LIN {X 0,Y 458.169,Z 588.59,A -85,B 0,C 180,E1 7423.789,E2 7423.789} C_VEL
LIN {X 0,Y 488.022,Z 647.13,A -85,B 0,C 180,E1 7427.64,E2 7427.64} C_VEL
LIN {X 0,Y 484.571,Z 716.932,A -85,B 0,C 180,E1 7429.58,E2 7429.58} C_VEL
LIN {X 0,Y 482.25,Z 744.899,A -85,B 0,C 180,E1 7430.929,E2 7430.929} C_VEL
LIN {X 0,Y 471.654,Z 776.533,A -85,B 0,C 180,E1 7432.394,E2 7432.394} C_VEL
LIN {X 0,Y 464.086,Z 836.053,A -85,B 0,C 180,E1 7437.824,E2 7437.824} C_VEL
LIN {X 0,Y 457.551,Z 880.34,A -85,B 0,C 180,E1 7444.194,E2 7444.194} C_VEL
LIN {X 0,Y 453.181,Z 916.717,A -85,B 0,C 180,E1 7452.427,E2 7452.427} C_VEL
LIN {X 0,Y 451.592,Z 937.285,A -85,B 0,C 180,E1 7460.326,E2 7460.326} C_VEL
LIN {X 0,Y 451.133,Z 945.148,A -85,B 0,C 180,E1 7467.107,E2 7467.107} C_VEL
LIN {X 0,Y 451.005,Z 943.768,A -85,B 0,C 180,E1 7474.824,E2 7474.824} C_VEL
LIN {X 0,Y 451.477,Z 931.075,A -85,B 0,C 180,E1 7482.619,E2 7482.619} C_VEL
LIN {X 0,Y 453.83,Z 905.664,A -85,B 0,C 180,E1 7490.554,E2 7490.554} C_VEL
LIN {X 0,Y 459.576,Z 865.156,A -85,B 0,C 180,E1 7498.336,E2 7498.336} C_VEL
LIN {X 0,Y 466.177,Z 818.816,A -85,B 0,C 180,E1 7503.99,E2 7503.99} C_VEL
LIN {X 0,Y 473.707,Z 757.778,A -85,B 0,C 180,E1 7508.771,E2 7508.771} C_VEL
LIN {X 0,Y 479.303,Z 694.506,A -85,B 0,C 180,E1 7511.694,E2 7511.694} C_VEL
LIN {X 0,Y 479.541,Z 644.153,A -85,B 0,C 180,E1 7512.988,E2 7512.988} C_VEL
LIN {X 0,Y 450.022,Z 586.94,A -85,B 0,C 180,E1 7516.817,E2 7516.817} C_VEL
LIN {X 0,Y 449.877,Z 586.94,A -85,B 0,C 180,E1 7526.24,E2 7526.24} C_VEL
LIN {X 0,Y 450.009,Z 586.94,A -85,B 0,C 180,E1 7535.12,E2 7535.12} C_VEL
LIN {X 0,Y 450.376,Z 586.94,A -85,B 0,C 180,E1 7545.406,E2 7545.406} C_VEL
LIN {X 0,Y 450.772,Z 586.94,A -85,B 0,C 180,E1 7555.211,E2 7555.211} C_VEL
LIN {X 0,Y 450.81,Z 586.94,A -85,B 0,C 180,E1 7562.93,E2 7562.93} C_VEL
LIN {X 0,Y 450.783,Z 586.94,A -85,B 0,C 180,E1 7572.672,E2 7572.672} C_VEL
LIN {X 0,Y 450.312,Z 586.94,A -85,B 0,C 180,E1 7582.832,E2 7582.832} C_VEL
LIN {X 0,Y 450.247,Z 588.263,A -85,B 0,C 180,E1 7593.002,E2 7593.002} C_VEL
LIN {X 0,Y 470.605,Z 632.247,A -85,B 0,C 180,E1 7595.934,E2 7595.934} C_VEL
LIN {X 0,Y 466.774,Z 687.738,A -85,B 0,C 180,E1 7598.161,E2 7598.161} C_VEL
LIN {X 0,Y 461.298,Z 735.974,A -85,B 0,C 180,E1 7602.044,E2 7602.044} C_VEL
LIN {X 0,Y 456.216,Z 774.865,A -85,B 0,C 180,E1 7607.473,E2 7607.473} C_VEL
LIN {X 0,Y 452.907,Z 801.492,A -85,B 0,C 180,E1 7614.102,E2 7614.102} C_VEL
LIN {X 0,Y 451.768,Z 813.36,A -85,B 0,C 180,E1 7620.853,E2 7620.853} C_VEL
LIN {X 0,Y 451.997,Z 812.735,A -85,B 0,C 180,E1 7627.45,E2 7627.45} C_VEL
LIN {X 0,Y 453.416,Z 798.561,A -85,B 0,C 180,E1 7634.471,E2 7634.471} C_VEL
LIN {X 0,Y 456.497,Z 770.469,A -85,B 0,C 180,E1 7640.916,E2 7640.916} C_VEL
LIN {X 0,Y 461.148,Z 730.969,A -85,B 0,C 180,E1 7646.109,E2 7646.109} C_VEL
LIN {X 0,Y 466.131,Z 680.829,A -85,B 0,C 180,E1 7649.884,E2 7649.884} C_VEL
LIN {X 0,Y 467.715,Z 623.987,A -85,B 0,C 180,E1 7652.015,E2 7652.015} C_VEL
LIN {X 0,Y 450.876,Z 586.94,A -85,B 0,C 180,E1 7654.344,E2 7654.344} C_VEL
LIN {X 0,Y 450.69,Z 586.94,A -85,B 0,C 180,E1 7664.628,E2 7664.628} C_VEL
LIN {X 0,Y 450.352,Z 586.94,A -85,B 0,C 180,E1 7674.912,E2 7674.912} C_VEL
LIN {X 0,Y 449.926,Z 586.94,A -85,B 0,C 180,E1 7684.243,E2 7684.243} C_VEL
LIN {X 0,Y 449.97,Z 586.94,A -85,B 0,C 180,E1 7693.739,E2 7693.739} C_VEL
LIN {X 0,Y 449.887,Z 586.94,A -85,B 0,C 180,E1 7703.793,E2 7703.793} C_VEL
LIN {X 0,Y 450.197,Z 586.94,A -85,B 0,C 180,E1 7713.288,E2 7713.288} C_VEL
LIN {X 0,Y 450.998,Z 586.94,A -85,B 0,C 180,E1 7725.351,E2 7725.351} C_VEL
LIN {X 0,Y 451.054,Z 586.94,A -85,B 0,C 180,E1 7735.14,E2 7735.14} C_VEL
LIN {X 0,Y 451.103,Z 586.94,A -85,B 0,C 180,E1 7742.854,E2 7742.854} C_VEL
LIN {X 0,Y 450.686,Z 586.94,A -85,B 0,C 180,E1 7752.599,E2 7752.599} C_VEL
LIN {X 0,Y 450.38,Z 586.94,A -85,B 0,C 180,E1 7762.748,E2 7762.748} C_VEL
LIN {X 0,Y 450.056,Z 586.94,A -85,B 0,C 180,E1 7771.452,E2 7771.452} C_VEL
LIN {X 0,Y 449.934,Z 586.94,A -85,B 0,C 180,E1 7781.055,E2 7781.055} C_VEL
LIN {X 0,Y 450.228,Z 588.983,A -85,B 0,C 180,E1 7782.975,E2 7782.975} C_VEL
LIN {X 0,Y 481.575,Z 650.873,A -85,B 0,C 180,E1 7787.149,E2 7787.149} C_VEL
LIN {X 0,Y 477.658,Z 720.311,A -85,B 0,C 180,E1 7789.193,E2 7789.193} C_VEL
LIN {X 0,Y 471.654,Z 776.533,A -85,B 0,C 180,E1 7792.394,E2 7792.394} C_VEL
LIN {X 0,Y 460.687,Z 806.318,A -85,B 0,C 180,E1 7794.355,E2 7794.355} C_VEL
LIN {X 0,Y 452.816,Z 861.229,A -85,B 0,C 180,E1 7800.634,E2 7800.634} C_VEL
LIN {X 0,Y 446.871,Z 900.269,A -85,B 0,C 180,E1 7807.802,E2 7807.802} C_VEL
LIN {X 0,Y 443.887,Z 927.251,A -85,B 0,C 180,E1 7815.616,E2 7815.616} C_VEL
LIN {X 0,Y 442.997,Z 941.682,A -85,B 0,C 180,E1 7823.113,E2 7823.113} C_VEL
LIN {X 0,Y 442.951,Z 945.837,A -85,B 0,C 180,E1 7830.981,E2 7830.981} C_VEL
LIN {X 0,Y 443.529,Z 938.888,A -85,B 0,C 180,E1 7838.856,E2 7838.856} C_VEL
LIN {X 0,Y 444.91,Z 918.74,A -85,B 0,C 180,E1 7847.306,E2 7847.306} C_VEL
LIN {X 0,Y 449.421,Z 883.452,A -85,B 0,C 180,E1 7855.689,E2 7855.689} C_VEL
LIN {X 0,Y 455.739,Z 841.528,A -85,B 0,C 180,E1 7861.897,E2 7861.897} C_VEL
LIN {X 0,Y 463.694,Z 782.474,A -85,B 0,C 180,E1 7867.571,E2 7867.571} C_VEL
LIN {X 0,Y 470.428,Z 717.472,A -85,B 0,C 180,E1 7871.397,E2 7871.397} C_VEL
LIN {X 0,Y 473.618,Z 648.362,A -85,B 0,C 180,E1 7873.423,E2 7873.423} C_VEL
LIN {X 0,Y 441.953,Z 586.94,A -85,B 0,C 180,E1 7877.646,E2 7877.646} C_VEL
LIN {X 0,Y 441.888,Z 586.94,A -85,B 0,C 180,E1 7887.898,E2 7887.898} C_VEL
LIN {X 0,Y 441.894,Z 586.94,A -85,B 0,C 180,E1 7896.789,E2 7896.789} C_VEL
LIN {X 0,Y 442.383,Z 586.94,A -85,B 0,C 180,E1 7907.16,E2 7907.16} C_VEL
LIN {X 0,Y 443.061,Z 586.94,A -85,B 0,C 180,E1 7917.094,E2 7917.094} C_VEL
LIN {X 0,Y 442.991,Z 586.94,A -85,B 0,C 180,E1 7926.921,E2 7926.921} C_VEL
LIN {X 0,Y 442.517,Z 586.94,A -85,B 0,C 180,E1 7936.979,E2 7936.979} C_VEL
LIN {X 0,Y 442.148,Z 586.94,A -85,B 0,C 180,E1 7947.633,E2 7947.633} C_VEL
LIN {X 0,Y 442.299,Z 588.447,A -85,B 0,C 180,E1 7952.157,E2 7952.157} C_VEL
LIN {X 0,Y 464.097,Z 633.334,A -85,B 0,C 180,E1 7955.381,E2 7955.381} C_VEL
LIN {X 0,Y 460.025,Z 688.479,A -85,B 0,C 180,E1 7957.637,E2 7957.637} C_VEL
LIN {X 0,Y 454.191,Z 736.885,A -85,B 0,C 180,E1 7961.585,E2 7961.585} C_VEL
LIN {X 0,Y 448.669,Z 776.328,A -85,B 0,C 180,E1 7967.192,E2 7967.192} C_VEL
LIN {X 0,Y 445.116,Z 802.915,A -85,B 0,C 180,E1 7973.971,E2 7973.971} C_VEL
LIN {X 0,Y 443.913,Z 814.525,A -85,B 0,C 180,E1 7980.695,E2 7980.695} C_VEL
LIN {X 0,Y 444.163,Z 813.367,A -85,B 0,C 180,E1 7988.071,E2 7988.071} C_VEL
LIN {X 0,Y 445.751,Z 798.121,A -85,B 0,C 180,E1 7995.208,E2 7995.208} C_VEL
LIN {X 0,Y 449.244,Z 768.674,A -85,B 0,C 180,E1 8001.747,E2 8001.747} C_VEL
LIN {X 0,Y 454.399,Z 728.304,A -85,B 0,C 180,E1 8006.89,E2 8006.89} C_VEL
LIN {X 0,Y 459.473,Z 677.695,A -85,B 0,C 180,E1 8010.592,E2 8010.592} C_VEL
LIN {X 0,Y 460.9,Z 626.072,A -85,B 0,C 180,E1 8012.536,E2 8012.536} C_VEL
LIN {X 0,Y 442.845,Z 586.94,A -85,B 0,C 180,E1 8015.125,E2 8015.125} C_VEL
LIN {X 0,Y 442.689,Z 586.94,A -85,B 0,C 180,E1 8024.899,E2 8024.899} C_VEL
LIN {X 0,Y 442.304,Z 586.94,A -85,B 0,C 180,E1 8035.397,E2 8035.397} C_VEL
LIN {X 0,Y 441.879,Z 586.94,A -85,B 0,C 180,E1 8046.159,E2 8046.159} C_VEL
LIN {X 0,Y 441.882,Z 586.94,A -85,B 0,C 180,E1 8055.22,E2 8055.22} C_VEL
LIN {X 0,Y 441.938,Z 586.94,A -85,B 0,C 180,E1 8065.458,E2 8065.458} C_VEL
LIN {X 0,Y 442.043,Z 586.94,A -85,B 0,C 180,E1 8075.471,E2 8075.471} C_VEL
LIN {X 0,Y 442.944,Z 586.94,A -85,B 0,C 180,E1 8085.078,E2 8085.078} C_VEL
LIN {X 0,Y 443.054,Z 586.94,A -85,B 0,C 180,E1 8095.052,E2 8095.052} C_VEL
LIN {X 0,Y 443.099,Z 586.94,A -85,B 0,C 180,E1 8102.906,E2 8102.906} C_VEL
LIN {X 0,Y 442.681,Z 586.94,A -85,B 0,C 180,E1 8112.831,E2 8112.831} C_VEL
LIN {X 0,Y 442.32,Z 586.94,A -85,B 0,C 180,E1 8123.187,E2 8123.187} C_VEL
LIN {X 0,Y 441.89,Z 586.94,A -85,B 0,C 180,E1 8132.714,E2 8132.714} C_VEL
LIN {X 0,Y 441.959,Z 587.932,A -85,B 0,C 180,E1 8142.056,E2 8142.056} C_VEL
LIN {X 0,Y 475.063,Z 653.403,A -85,B 0,C 180,E1 8146.623,E2 8146.623} C_VEL
LIN {X 0,Y 470.893,Z 721.885,A -85,B 0,C 180,E1 8148.715,E2 8148.715} C_VEL
LIN {X 0,Y 463.303,Z 786.983,A -85,B 0,C 180,E1 8152.701,E2 8152.701} C_VEL
LIN {X 0,Y 460.687,Z 806.318,A -85,B 0,C 180,E1 8154.355,E2 8154.355} C_VEL
LIN {X 0,Y 449.477,Z 833.905,A -85,B 0,C 180,E1 8156.789,E2 8156.789} C_VEL
LIN {X 0,Y 442.059,Z 883.424,A -85,B 0,C 180,E1 8163.885,E2 8163.885} C_VEL
LIN {X 0,Y 437.357,Z 917.884,A -85,B 0,C 180,E1 8172.12,E2 8172.12} C_VEL
LIN {X 0,Y 435.342,Z 938.885,A -85,B 0,C 180,E1 8180.974,E2 8180.974} C_VEL
LIN {X 0,Y 434.71,Z 945.836,A -85,B 0,C 180,E1 8188.999,E2 8188.999} C_VEL
LIN {X 0,Y 435.04,Z 942.008,A -85,B 0,C 180,E1 8196.743,E2 8196.743} C_VEL
LIN {X 0,Y 436.422,Z 926.004,A -85,B 0,C 180,E1 8205.116,E2 8205.116} C_VEL
LIN {X 0,Y 440.39,Z 894.795,A -85,B 0,C 180,E1 8213.821,E2 8213.821} C_VEL
LIN {X 0,Y 446.363,Z 853.79,A -85,B 0,C 180,E1 8220.676,E2 8220.676} C_VEL
LIN {X 0,Y 454.368,Z 798.67,A -85,B 0,C 180,E1 8226.717,E2 8226.717} C_VEL
LIN {X 0,Y 462.395,Z 734.002,A -85,B 0,C 180,E1 8231.145,E2 8231.145} C_VEL
LIN {X 0,Y 467.756,Z 665.782,A -85,B 0,C 180,E1 8233.565,E2 8233.565} C_VEL
LIN {X 0,Y 466.044,Z 649.71,A -85,B 0,C 180,E1 8234.069,E2 8234.069} C_VEL
LIN {X 0,Y 433.804,Z 586.94,A -85,B 0,C 180,E1 8238.772,E2 8238.772} C_VEL
LIN {X 0,Y 433.883,Z 586.94,A -85,B 0,C 180,E1 8249.584,E2 8249.584} C_VEL
LIN {X 0,Y 434.034,Z 586.94,A -85,B 0,C 180,E1 8260.649,E2 8260.649} C_VEL
LIN {X 0,Y 434.788,Z 586.94,A -85,B 0,C 180,E1 8271.006,E2 8271.006} C_VEL
LIN {X 0,Y 434.99,Z 586.94,A -85,B 0,C 180,E1 8281.037,E2 8281.037} C_VEL
LIN {X 0,Y 434.689,Z 586.94,A -85,B 0,C 180,E1 8291.104,E2 8291.104} C_VEL
LIN {X 0,Y 434.312,Z 586.94,A -85,B 0,C 180,E1 8301.555,E2 8301.555} C_VEL
LIN {X 0,Y 434.283,Z 588.609,A -85,B 0,C 180,E1 8311.257,E2 8311.257} C_VEL
LIN {X 0,Y 457.496,Z 636.351,A -85,B 0,C 180,E1 8314.86,E2 8314.86} C_VEL
LIN {X 0,Y 453.064,Z 691.771,A -85,B 0,C 180,E1 8317.248,E2 8317.248} C_VEL
LIN {X 0,Y 446.787,Z 740.13,A -85,B 0,C 180,E1 8321.372,E2 8321.372} C_VEL
LIN {X 0,Y 440.994,Z 778.652,A -85,B 0,C 180,E1 8327.07,E2 8327.07} C_VEL
LIN {X 0,Y 437.367,Z 804.102,A -85,B 0,C 180,E1 8333.742,E2 8333.742} C_VEL
LIN {X 0,Y 436.213,Z 814.929,A -85,B 0,C 180,E1 8339.707,E2 8339.707} C_VEL
LIN {X 0,Y 436.15,Z 815.44,A -85,B 0,C 180,E1 8347.268,E2 8347.268} C_VEL
LIN {X 0,Y 437.655,Z 802.32,A -85,B 0,C 180,E1 8354.413,E2 8354.413} C_VEL
LIN {X 0,Y 441.131,Z 775.355,A -85,B 0,C 180,E1 8361.096,E2 8361.096} C_VEL
LIN {X 0,Y 446.278,Z 736.498,A -85,B 0,C 180,E1 8366.589,E2 8366.589} C_VEL
LIN {X 0,Y 451.94,Z 687.345,A -85,B 0,C 180,E1 8370.602,E2 8370.602} C_VEL
LIN {X 0,Y 454.589,Z 629.258,A -85,B 0,C 180,E1 8373.005,E2 8373.005} C_VEL
LIN {X 0,Y 434.847,Z 586.94,A -85,B 0,C 180,E1 8376.013,E2 8376.013} C_VEL
LIN {X 0,Y 434.603,Z 586.94,A -85,B 0,C 180,E1 8386.156,E2 8386.156} C_VEL
LIN {X 0,Y 434.145,Z 586.94,A -85,B 0,C 180,E1 8396.92,E2 8396.92} C_VEL
LIN {X 0,Y 433.783,Z 586.94,A -85,B 0,C 180,E1 8407.75,E2 8407.75} C_VEL
LIN {X 0,Y 433.843,Z 586.94,A -85,B 0,C 180,E1 8416.963,E2 8416.963} C_VEL
LIN {X 0,Y 433.937,Z 586.94,A -85,B 0,C 180,E1 8427.146,E2 8427.146} C_VEL
LIN {X 0,Y 433.974,Z 586.94,A -85,B 0,C 180,E1 8436.257,E2 8436.257} C_VEL
LIN {X 0,Y 434.948,Z 586.94,A -85,B 0,C 180,E1 8446.858,E2 8446.858} C_VEL
LIN {X 0,Y 434.869,Z 586.94,A -85,B 0,C 180,E1 8456.963,E2 8456.963} C_VEL
LIN {X 0,Y 434.844,Z 586.94,A -85,B 0,C 180,E1 8465.953,E2 8465.953} C_VEL
LIN {X 0,Y 434.542,Z 586.94,A -85,B 0,C 180,E1 8476.183,E2 8476.183} C_VEL
LIN {X 0,Y 434.1,Z 586.94,A -85,B 0,C 180,E1 8486.945,E2 8486.945} C_VEL
LIN {X 0,Y 433.789,Z 586.94,A -85,B 0,C 180,E1 8498.082,E2 8498.082} C_VEL
LIN {X 0,Y 434.037,Z 588.819,A -85,B 0,C 180,E1 8501.182,E2 8501.182} C_VEL
LIN {X 0,Y 468.637,Z 655.096,A -85,B 0,C 180,E1 8506.07,E2 8506.07} C_VEL
LIN {X 0,Y 464.129,Z 723.218,A -85,B 0,C 180,E1 8508.216,E2 8508.216} C_VEL
LIN {X 0,Y 455.937,Z 789.536,A -85,B 0,C 180,E1 8512.408,E2 8512.408} C_VEL
LIN {X 0,Y 449.477,Z 833.905,A -85,B 0,C 180,E1 8516.789,E2 8516.789} C_VEL
LIN {X 0,Y 437.861,Z 859.062,A -85,B 0,C 180,E1 8519.666,E2 8519.666} C_VEL
LIN {X 0,Y 431.186,Z 902.39,A -85,B 0,C 180,E1 8527.496,E2 8527.496} C_VEL
LIN {X 0,Y 427.932,Z 928.676,A -85,B 0,C 180,E1 8535.626,E2 8535.626} C_VEL
LIN {X 0,Y 427.026,Z 941.682,A -85,B 0,C 180,E1 8542.854,E2 8542.854} C_VEL
LIN {X 0,Y 426.968,Z 945.836,A -85,B 0,C 180,E1 8551.017,E2 8551.017} C_VEL
LIN {X 0,Y 427.545,Z 938.888,A -85,B 0,C 180,E1 8559.19,E2 8559.19} C_VEL
LIN {X 0,Y 429.126,Z 918.103,A -85,B 0,C 180,E1 8568.167,E2 8568.167} C_VEL
LIN {X 0,Y 433.56,Z 887.265,A -85,B 0,C 180,E1 8575.634,E2 8575.634} C_VEL
LIN {X 0,Y 441.327,Z 837.188,A -85,B 0,C 180,E1 8583.171,E2 8583.171} C_VEL
LIN {X 0,Y 450.385,Z 777.063,A -85,B 0,C 180,E1 8588.963,E2 8588.963} C_VEL
LIN {X 0,Y 457.8,Z 711.447,A -85,B 0,C 180,E1 8592.742,E2 8592.742} C_VEL
LIN {X 0,Y 459.92,Z 653.52,A -85,B 0,C 180,E1 8594.552,E2 8594.552} C_VEL
LIN {X 0,Y 425.793,Z 586.94,A -85,B 0,C 180,E1 8599.788,E2 8599.788} C_VEL
LIN {X 0,Y 425.844,Z 586.94,A -85,B 0,C 180,E1 8610.816,E2 8610.816} C_VEL
LIN {X 0,Y 426.057,Z 586.94,A -85,B 0,C 180,E1 8620.709,E2 8620.709} C_VEL
LIN {X 0,Y 426.74,Z 586.94,A -85,B 0,C 180,E1 8630.835,E2 8630.835} C_VEL
LIN {X 0,Y 426.983,Z 586.94,A -85,B 0,C 180,E1 8641.057,E2 8641.057} C_VEL
LIN {X 0,Y 426.665,Z 586.94,A -85,B 0,C 180,E1 8651.316,E2 8651.316} C_VEL
LIN {X 0,Y 426.273,Z 586.94,A -85,B 0,C 180,E1 8661.983,E2 8661.983} C_VEL
LIN {X 0,Y 426.248,Z 588.66,A -85,B 0,C 180,E1 8670.3,E2 8670.3} C_VEL
LIN {X 0,Y 450.946,Z 639.816,A -85,B 0,C 180,E1 8674.344,E2 8674.344} C_VEL
LIN {X 0,Y 446.189,Z 694.336,A -85,B 0,C 180,E1 8676.808,E2 8676.808} C_VEL
LIN {X 0,Y 439.283,Z 743.687,A -85,B 0,C 180,E1 8681.18,E2 8681.18} C_VEL
LIN {X 0,Y 433.078,Z 782.406,A -85,B 0,C 180,E1 8687.226,E2 8687.226} C_VEL
LIN {X 0,Y 429.337,Z 807.304,A -85,B 0,C 180,E1 8694.325,E2 8694.325} C_VEL
LIN {X 0,Y 428.01,Z 817.628,A -85,B 0,C 180,E1 8701.404,E2 8701.404} C_VEL
LIN {X 0,Y 428.517,Z 814.776,A -85,B 0,C 180,E1 8709.075,E2 8709.075} C_VEL
LIN {X 0,Y 430.294,Z 798.637,A -85,B 0,C 180,E1 8716.215,E2 8716.215} C_VEL
LIN {X 0,Y 434.43,Z 769.3,A -85,B 0,C 180,E1 8722.726,E2 8722.726} C_VEL
LIN {X 0,Y 440.48,Z 727.432,A -85,B 0,C 180,E1 8728.079,E2 8728.079} C_VEL
LIN {X 0,Y 446.179,Z 676.478,A -85,B 0,C 180,E1 8731.779,E2 8731.779} C_VEL
LIN {X 0,Y 447.559,Z 630.648,A -85,B 0,C 180,E1 8733.599,E2 8733.599} C_VEL
LIN {X 0,Y 426.931,Z 586.94,A -85,B 0,C 180,E1 8736.749,E2 8736.749} C_VEL
LIN {X 0,Y 426.524,Z 586.94,A -85,B 0,C 180,E1 8747.604,E2 8747.604} C_VEL
LIN {X 0,Y 426.042,Z 586.94,A -85,B 0,C 180,E1 8758.742,E2 8758.742} C_VEL
LIN {X 0,Y 425.769,Z 586.94,A -85,B 0,C 180,E1 8769.944,E2 8769.944} C_VEL
LIN {X 0,Y 425.751,Z 586.94,A -85,B 0,C 180,E1 8780.027,E2 8780.027} C_VEL
LIN {X 0,Y 425.934,Z 586.94,A -85,B 0,C 180,E1 8790.798,E2 8790.798} C_VEL
LIN {X 0,Y 426.43,Z 586.94,A -85,B 0,C 180,E1 8802.359,E2 8802.359} C_VEL
LIN {X 0,Y 427.02,Z 586.94,A -85,B 0,C 180,E1 8812.819,E2 8812.819} C_VEL
LIN {X 0,Y 427.065,Z 586.94,A -85,B 0,C 180,E1 8823.015,E2 8823.015} C_VEL
LIN {X 0,Y 426.616,Z 586.94,A -85,B 0,C 180,E1 8833.323,E2 8833.323} C_VEL
LIN {X 0,Y 426.211,Z 586.94,A -85,B 0,C 180,E1 8844.118,E2 8844.118} C_VEL
LIN {X 0,Y 425.824,Z 586.94,A -85,B 0,C 180,E1 8853.468,E2 8853.468} C_VEL
LIN {X 0,Y 426.061,Z 588.944,A -85,B 0,C 180,E1 8860.243,E2 8860.243} C_VEL
LIN {X 0,Y 462.209,Z 659.065,A -85,B 0,C 180,E1 8865.551,E2 8865.551} C_VEL
LIN {X 0,Y 457.276,Z 725.665,A -85,B 0,C 180,E1 8867.767,E2 8867.767} C_VEL
LIN {X 0,Y 448.796,Z 790.205,A -85,B 0,C 180,E1 8871.959,E2 8871.959} C_VEL
LIN {X 0,Y 439.619,Z 848.816,A -85,B 0,C 180,E1 8878.235,E2 8878.235} C_VEL
LIN {X 0,Y 437.861,Z 859.062,A -85,B 0,C 180,E1 8879.666,E2 8879.666} C_VEL
LIN {X 0,Y 426.697,Z 881.341,A -85,B 0,C 180,E1 8883.017,E2 8883.017} C_VEL
LIN {X 0,Y 421.594,Z 916.8,A -85,B 0,C 180,E1 8891.097,E2 8891.097} C_VEL
LIN {X 0,Y 419.698,Z 937.285,A -85,B 0,C 180,E1 8899.583,E2 8899.583} C_VEL
LIN {X 0,Y 419.173,Z 945.146,A -85,B 0,C 180,E1 8906.886,E2 8906.886} C_VEL
LIN {X 0,Y 418.994,Z 943.279,A -85,B 0,C 180,E1 8915.783,E2 8915.783} C_VEL
LIN {X 0,Y 420.239,Z 928.682,A -85,B 0,C 180,E1 8924.641,E2 8924.641} C_VEL
LIN {X 0,Y 423.518,Z 902.321,A -85,B 0,C 180,E1 8932.654,E2 8932.654} C_VEL
LIN {X 0,Y 430.369,Z 858.093,A -85,B 0,C 180,E1 8940.748,E2 8940.748} C_VEL
LIN {X 0,Y 439.664,Z 800.966,A -85,B 0,C 180,E1 8947.467,E2 8947.467} C_VEL
LIN {X 0,Y 448.65,Z 736.587,A -85,B 0,C 180,E1 8952.116,E2 8952.116} C_VEL
LIN {X 0,Y 454.609,Z 671.773,A -85,B 0,C 180,E1 8954.597,E2 8954.597} C_VEL
LIN {X 0,Y 452.871,Z 655.597,A -85,B 0,C 180,E1 8955.182,E2 8955.182} C_VEL
LIN {X 0,Y 419.043,Z 591.318,A -85,B 0,C 180,E1 8960.277,E2 8960.277} C_VEL
LIN {X 0,Y 417.708,Z 586.94,A -85,B 0,C 180,E1 8960.593,E2 8960.593} C_VEL
LIN {X 0,Y 417.848,Z 586.94,A -85,B 0,C 180,E1 8970.699,E2 8970.699} C_VEL
LIN {X 0,Y 418.109,Z 586.94,A -85,B 0,C 180,E1 8982.08,E2 8982.08} C_VEL
LIN {X 0,Y 418.83,Z 586.94,A -85,B 0,C 180,E1 8992.757,E2 8992.757} C_VEL
LIN {X 0,Y 418.977,Z 586.94,A -85,B 0,C 180,E1 9001.077,E2 9001.077} C_VEL
LIN {X 0,Y 418.667,Z 586.94,A -85,B 0,C 180,E1 9011.535,E2 9011.535} C_VEL
LIN {X 0,Y 418.21,Z 586.94,A -85,B 0,C 180,E1 9022.429,E2 9022.429} C_VEL
LIN {X 0,Y 418.249,Z 588.819,A -85,B 0,C 180,E1 9029.29,E2 9029.29} C_VEL
LIN {X 0,Y 444.534,Z 641.378,A -85,B 0,C 180,E1 9033.754,E2 9033.754} C_VEL
LIN {X 0,Y 439.391,Z 696.31,A -85,B 0,C 180,E1 9036.318,E2 9036.318} C_VEL
LIN {X 0,Y 432.088,Z 745.649,A -85,B 0,C 180,E1 9040.808,E2 9040.808} C_VEL
LIN {X 0,Y 425.485,Z 784.313,A -85,B 0,C 180,E1 9047.015,E2 9047.015} C_VEL
LIN {X 0,Y 421.578,Z 808.562,A -85,B 0,C 180,E1 9054.123,E2 9054.123} C_VEL
LIN {X 0,Y 420.19,Z 818.508,A -85,B 0,C 180,E1 9060.821,E2 9060.821} C_VEL
LIN {X 0,Y 420.371,Z 817.591,A -85,B 0,C 180,E1 9067.726,E2 9067.726} C_VEL
LIN {X 0,Y 422.196,Z 804.072,A -85,B 0,C 180,E1 9075.039,E2 9075.039} C_VEL
LIN {X 0,Y 426.26,Z 776.084,A -85,B 0,C 180,E1 9082.072,E2 9082.072} C_VEL
LIN {X 0,Y 432.361,Z 735.931,A -85,B 0,C 180,E1 9087.777,E2 9087.777} C_VEL
LIN {X 0,Y 438.654,Z 685.673,A -85,B 0,C 180,E1 9091.859,E2 9091.859} C_VEL
LIN {X 0,Y 441.138,Z 633.549,A -85,B 0,C 180,E1 9094.12,E2 9094.12} C_VEL
LIN {X 0,Y 418.876,Z 586.94,A -85,B 0,C 180,E1 9097.809,E2 9097.809} C_VEL
LIN {X 0,Y 418.484,Z 586.94,A -85,B 0,C 180,E1 9107.954,E2 9107.954} C_VEL
LIN {X 0,Y 418.074,Z 586.94,A -85,B 0,C 180,E1 9117.172,E2 9117.172} C_VEL
LIN {X 0,Y 417.744,Z 586.94,A -85,B 0,C 180,E1 9128.611,E2 9128.611} C_VEL
LIN {X 0,Y 417.806,Z 586.94,A -85,B 0,C 180,E1 9138.125,E2 9138.125} C_VEL
LIN {X 0,Y 417.896,Z 586.94,A -85,B 0,C 180,E1 9148.581,E2 9148.581} C_VEL
LIN {X 0,Y 417.994,Z 586.94,A -85,B 0,C 180,E1 9159.791,E2 9159.791} C_VEL
LIN {X 0,Y 418.803,Z 586.94,A -85,B 0,C 180,E1 9168.469,E2 9168.469} C_VEL
LIN {X 0,Y 419.029,Z 586.94,A -85,B 0,C 180,E1 9179.027,E2 9179.027} C_VEL
LIN {X 0,Y 418.863,Z 586.94,A -85,B 0,C 180,E1 9189.339,E2 9189.339} C_VEL
LIN {X 0,Y 418.306,Z 586.94,A -85,B 0,C 180,E1 9200.109,E2 9200.109} C_VEL
LIN {X 0,Y 417.881,Z 586.94,A -85,B 0,C 180,E1 9211.415,E2 9211.415} C_VEL
LIN {X 0,Y 417.901,Z 588.507,A -85,B 0,C 180,E1 9219.229,E2 9219.229} C_VEL
LIN {X 0,Y 455.863,Z 659.832,A -85,B 0,C 180,E1 9224.949,E2 9224.949} C_VEL
LIN {X 0,Y 450.684,Z 725.701,A -85,B 0,C 180,E1 9227.183,E2 9227.183} C_VEL
LIN {X 0,Y 441.848,Z 789.565,A -85,B 0,C 180,E1 9231.381,E2 9231.381} C_VEL
LIN {X 0,Y 432.357,Z 847.239,A -85,B 0,C 180,E1 9237.638,E2 9237.638} C_VEL
LIN {X 0,Y 426.697,Z 881.341,A -85,B 0,C 180,E1 9243.017,E2 9243.017} C_VEL
LIN {X 0,Y 415.654,Z 900.633,A -85,B 0,C 180,E1 9246.804,E2 9246.804} C_VEL
LIN {X 0,Y 412.178,Z 928.621,A -85,B 0,C 180,E1 9255.064,E2 9255.064} C_VEL
LIN {X 0,Y 411.059,Z 941.681,A -85,B 0,C 180,E1 9262.575,E2 9262.575} C_VEL
LIN {X 0,Y 410.971,Z 945.836,A -85,B 0,C 180,E1 9271.057,E2 9271.057} C_VEL
LIN {X 0,Y 411.546,Z 938.888,A -85,B 0,C 180,E1 9279.55,E2 9279.55} C_VEL
LIN {X 0,Y 413.124,Z 920.966,A -85,B 0,C 180,E1 9287.644,E2 9287.644} C_VEL
LIN {X 0,Y 418.036,Z 885.409,A -85,B 0,C 180,E1 9296.402,E2 9296.402} C_VEL
LIN {X 0,Y 426.669,Z 835.274,A -85,B 0,C 180,E1 9304.221,E2 9304.221} C_VEL
LIN {X 0,Y 436.786,Z 774.672,A -85,B 0,C 180,E1 9310.204,E2 9310.204} C_VEL
LIN {X 0,Y 444.904,Z 709.56,A -85,B 0,C 180,E1 9314,E2 9314} C_VEL
LIN {X 0,Y 447.168,Z 659.93,A -85,B 0,C 180,E1 9315.653,E2 9315.653} C_VEL
LIN {X 0,Y 414.497,Z 596.884,A -85,B 0,C 180,E1 9320.759,E2 9320.759} C_VEL
LIN {X 0,Y 409.68,Z 586.94,A -85,B 0,C 180,E1 9321.932,E2 9321.932} C_VEL
LIN {X 0,Y 409.823,Z 586.94,A -85,B 0,C 180,E1 9332.486,E2 9332.486} C_VEL
LIN {X 0,Y 410.218,Z 586.94,A -85,B 0,C 180,E1 9343.941,E2 9343.941} C_VEL
LIN {X 0,Y 410.778,Z 586.94,A -85,B 0,C 180,E1 9354.743,E2 9354.743} C_VEL
LIN {X 0,Y 410.861,Z 586.94,A -85,B 0,C 180,E1 9363.215,E2 9363.215} C_VEL
LIN {X 0,Y 410.582,Z 586.94,A -85,B 0,C 180,E1 9373.937,E2 9373.937} C_VEL
LIN {X 0,Y 410.067,Z 586.94,A -85,B 0,C 180,E1 9385.221,E2 9385.221} C_VEL
LIN {X 0,Y 410.139,Z 588.424,A -85,B 0,C 180,E1 9388.182,E2 9388.182} C_VEL
LIN {X 0,Y 438.09,Z 644.461,A -85,B 0,C 180,E1 9393.192,E2 9393.192} C_VEL
LIN {X 0,Y 432.594,Z 698.727,A -85,B 0,C 180,E1 9395.843,E2 9395.843} C_VEL
LIN {X 0,Y 424.915,Z 747.376,A -85,B 0,C 180,E1 9400.395,E2 9400.395} C_VEL
LIN {X 0,Y 418.037,Z 785.426,A -85,B 0,C 180,E1 9406.627,E2 9406.627} C_VEL
LIN {X 0,Y 413.796,Z 809.916,A -85,B 0,C 180,E1 9413.952,E2 9413.952} C_VEL
LIN {X 0,Y 412.429,Z 819.356,A -85,B 0,C 180,E1 9420.217,E2 9420.217} C_VEL
LIN {X 0,Y 412.612,Z 818.191,A -85,B 0,C 180,E1 9428.422,E2 9428.422} C_VEL
LIN {X 0,Y 414.697,Z 802.481,A -85,B 0,C 180,E1 9436.241,E2 9436.241} C_VEL
LIN {X 0,Y 419.356,Z 772.608,A -85,B 0,C 180,E1 9443.29,E2 9443.29} C_VEL
LIN {X 0,Y 426.105,Z 731.1,A -85,B 0,C 180,E1 9448.872,E2 9448.872} C_VEL
LIN {X 0,Y 432.485,Z 680.501,A -85,B 0,C 180,E1 9452.766,E2 9452.766} C_VEL
LIN {X 0,Y 434.419,Z 635.352,A -85,B 0,C 180,E1 9454.708,E2 9454.708} C_VEL
LIN {X 0,Y 410.889,Z 586.94,A -85,B 0,C 180,E1 9458.496,E2 9458.496} C_VEL
LIN {X 0,Y 410.363,Z 586.94,A -85,B 0,C 180,E1 9469.384,E2 9469.384} C_VEL
LIN {X 0,Y 409.941,Z 586.94,A -85,B 0,C 180,E1 9479.984,E2 9479.984} C_VEL
LIN {X 0,Y 409.688,Z 586.94,A -85,B 0,C 180,E1 9490.559,E2 9490.559} C_VEL
LIN {X 0,Y 409.676,Z 586.94,A -85,B 0,C 180,E1 9499.558,E2 9499.558} C_VEL
LIN {X 0,Y 409.924,Z 586.94,A -85,B 0,C 180,E1 9510.456,E2 9510.456} C_VEL
LIN {X 0,Y 410.237,Z 586.94,A -85,B 0,C 180,E1 9521.639,E2 9521.639} C_VEL
LIN {X 0,Y 410.748,Z 586.94,A -85,B 0,C 180,E1 9530.393,E2 9530.393} C_VEL
LIN {X 0,Y 411.484,Z 586.94,A -85,B 0,C 180,E1 9541.016,E2 9541.016} C_VEL
LIN {X 0,Y 410.654,Z 586.94,A -85,B 0,C 180,E1 9551.681,E2 9551.681} C_VEL
LIN {X 0,Y 410.17,Z 586.94,A -85,B 0,C 180,E1 9562.806,E2 9562.806} C_VEL
LIN {X 0,Y 409.697,Z 586.94,A -85,B 0,C 180,E1 9573.549,E2 9573.549} C_VEL
LIN {X 0,Y 409.977,Z 588.888,A -85,B 0,C 180,E1 9578.213,E2 9578.213} C_VEL
LIN {X 0,Y 449.242,Z 662.365,A -85,B 0,C 180,E1 9584.343,E2 9584.343} C_VEL
LIN {X 0,Y 443.696,Z 729.724,A -85,B 0,C 180,E1 9586.785,E2 9586.785} C_VEL
LIN {X 0,Y 434.261,Z 793.271,A -85,B 0,C 180,E1 9591.184,E2 9591.184} C_VEL
LIN {X 0,Y 424.46,Z 849.399,A -85,B 0,C 180,E1 9597.542,E2 9597.542} C_VEL
LIN {X 0,Y 416.725,Z 895.06,A -85,B 0,C 180,E1 9605.529,E2 9605.529} C_VEL
LIN {X 0,Y 415.654,Z 900.633,A -85,B 0,C 180,E1 9606.804,E2 9606.804} C_VEL
LIN {X 0,Y 405.629,Z 916.602,A -85,B 0,C 180,E1 9611.001,E2 9611.001} C_VEL
LIN {X 0,Y 403.503,Z 938.793,A -85,B 0,C 180,E1 9620.255,E2 9620.255} C_VEL
LIN {X 0,Y 402.753,Z 945.835,A -85,B 0,C 180,E1 9628.92,E2 9628.92} C_VEL
LIN {X 0,Y 403.212,Z 941.683,A -85,B 0,C 180,E1 9637.568,E2 9637.568} C_VEL
LIN {X 0,Y 404.936,Z 924.509,A -85,B 0,C 180,E1 9646.323,E2 9646.323} C_VEL
LIN {X 0,Y 409.46,Z 890.645,A -85,B 0,C 180,E1 9655.52,E2 9655.52} C_VEL
LIN {X 0,Y 417.683,Z 844.046,A -85,B 0,C 180,E1 9663.479,E2 9663.479} C_VEL
LIN {X 0,Y 427.883,Z 786.659,A -85,B 0,C 180,E1 9669.78,E2 9669.78} C_VEL
LIN {X 0,Y 436.937,Z 721.843,A -85,B 0,C 180,E1 9674.082,E2 9674.082} C_VEL
LIN {X 0,Y 440.867,Z 663.007,A -85,B 0,C 180,E1 9676.228,E2 9676.228} C_VEL
LIN {X 0,Y 409.714,Z 602.031,A -85,B 0,C 180,E1 9681.301,E2 9681.301} C_VEL
LIN {X 0,Y 401.659,Z 586.94,A -85,B 0,C 180,E1 9683.114,E2 9683.114} C_VEL
LIN {X 0,Y 401.776,Z 586.94,A -85,B 0,C 180,E1 9694.312,E2 9694.312} C_VEL
LIN {X 0,Y 402.217,Z 586.94,A -85,B 0,C 180,E1 9705.852,E2 9705.852} C_VEL
LIN {X 0,Y 402.993,Z 586.94,A -85,B 0,C 180,E1 9716.804,E2 9716.804} C_VEL
LIN {X 0,Y 402.83,Z 586.94,A -85,B 0,C 180,E1 9727.615,E2 9727.615} C_VEL
LIN {X 0,Y 402.29,Z 586.94,A -85,B 0,C 180,E1 9738.737,E2 9738.737} C_VEL
LIN {X 0,Y 402.145,Z 588.625,A -85,B 0,C 180,E1 9747.03,E2 9747.03} C_VEL
LIN {X 0,Y 431.699,Z 645.152,A -85,B 0,C 180,E1 9752.522,E2 9752.522} C_VEL
LIN {X 0,Y 425.809,Z 701.384,A -85,B 0,C 180,E1 9755.369,E2 9755.369} C_VEL
LIN {X 0,Y 417.764,Z 749.252,A -85,B 0,C 180,E1 9759.983,E2 9759.983} C_VEL
LIN {X 0,Y 410.717,Z 786.094,A -85,B 0,C 180,E1 9766.129,E2 9766.129} C_VEL
LIN {X 0,Y 406.109,Z 810.624,A -85,B 0,C 180,E1 9773.493,E2 9773.493} C_VEL
LIN {X 0,Y 404.713,Z 820.18,A -85,B 0,C 180,E1 9779.59,E2 9779.59} C_VEL
LIN {X 0,Y 404.621,Z 819.904,A -85,B 0,C 180,E1 9788.01,E2 9788.01} C_VEL
LIN {X 0,Y 406.81,Z 805.109,A -85,B 0,C 180,E1 9795.969,E2 9795.969} C_VEL
LIN {X 0,Y 411.561,Z 776.423,A -85,B 0,C 180,E1 9803.177,E2 9803.177} C_VEL
LIN {X 0,Y 418.553,Z 735.998,A -85,B 0,C 180,E1 9808.962,E2 9808.962} C_VEL
LIN {X 0,Y 425.468,Z 684.888,A -85,B 0,C 180,E1 9813.142,E2 9813.142} C_VEL
LIN {X 0,Y 427.84,Z 637.697,A -85,B 0,C 180,E1 9815.285,E2 9815.285} C_VEL
LIN {X 0,Y 402.858,Z 586.94,A -85,B 0,C 180,E1 9819.46,E2 9819.46} C_VEL
LIN {X 0,Y 402.384,Z 586.94,A -85,B 0,C 180,E1 9828.698,E2 9828.698} C_VEL
LIN {X 0,Y 401.967,Z 586.94,A -85,B 0,C 180,E1 9838.159,E2 9838.159} C_VEL
LIN {X 0,Y 401.588,Z 586.94,A -85,B 0,C 180,E1 9849.189,E2 9849.189} C_VEL
LIN {X 0,Y 401.594,Z 586.94,A -85,B 0,C 180,E1 9858.568,E2 9858.568} C_VEL
LIN {X 0,Y 401.779,Z 586.94,A -85,B 0,C 180,E1 9869.309,E2 9869.309} C_VEL
LIN {X 0,Y 401.883,Z 586.94,A -85,B 0,C 180,E1 9878.943,E2 9878.943} C_VEL
LIN {X 0,Y 402.812,Z 586.94,A -85,B 0,C 180,E1 9888.004,E2 9888.004} C_VEL
LIN {X 0,Y 403.037,Z 586.94,A -85,B 0,C 180,E1 9899.057,E2 9899.057} C_VEL
LIN {X 0,Y 402.793,Z 586.94,A -85,B 0,C 180,E1 9909.715,E2 9909.715} C_VEL
LIN {X 0,Y 402.195,Z 586.94,A -85,B 0,C 180,E1 9920.952,E2 9920.952} C_VEL
LIN {X 0,Y 401.696,Z 586.94,A -85,B 0,C 180,E1 9931.787,E2 9931.787} C_VEL
LIN {X 0,Y 401.994,Z 588.943,A -85,B 0,C 180,E1 9937.135,E2 9937.135} C_VEL
LIN {X 0,Y 439.888,Z 659.439,A -85,B 0,C 180,E1 9943.298,E2 9943.298} C_VEL
LIN {X 0,Y 442.843,Z 670.948,A -85,B 0,C 180,E1 9943.943,E2 9943.943} C_VEL
LIN {X 0,Y 436.485,Z 735.383,A -85,B 0,C 180,E1 9946.469,E2 9946.469} C_VEL
LIN {X 0,Y 426.301,Z 799.032,A -85,B 0,C 180,E1 9951.169,E2 9951.169} C_VEL
LIN {X 0,Y 416.03,Z 854.149,A -85,B 0,C 180,E1 9957.834,E2 9957.834} C_VEL
LIN {X 0,Y 408.152,Z 898.282,A -85,B 0,C 180,E1 9966.108,E2 9966.108} C_VEL
LIN {X 0,Y 405.629,Z 916.602,A -85,B 0,C 180,E1 9971.001,E2 9971.001} C_VEL
LIN {X 0,Y 396.046,Z 928.889,A -85,B 0,C 180,E1 9975.587,E2 9975.587} C_VEL
LIN {X 0,Y 395.204,Z 943.097,A -85,B 0,C 180,E1 9984.49,E2 9984.49} C_VEL
LIN {X 0,Y 395.274,Z 944.67,A -85,B 0,C 180,E1 9993.3,E2 9993.3} C_VEL
LIN {X 0,Y 395.659,Z 933.605,A -85,B 0,C 180,E1 10002.177,E2 10002.177} C_VEL
LIN {X 0,Y 398.038,Z 910.807,A -85,B 0,C 180,E1 10010.649,E2 10010.649} C_VEL
LIN {X 0,Y 404.356,Z 873.339,A -85,B 0,C 180,E1 10019.2,E2 10019.2} C_VEL
LIN {X 0,Y 414.35,Z 822.004,A -85,B 0,C 180,E1 10026.74,E2 10026.74} C_VEL
LIN {X 0,Y 425.247,Z 761.058,A -85,B 0,C 180,E1 10032.355,E2 10032.355} C_VEL
LIN {X 0,Y 433.353,Z 699.091,A -85,B 0,C 180,E1 10035.654,E2 10035.654} C_VEL
LIN {X 0,Y 434.533,Z 666.012,A -85,B 0,C 180,E1 10036.81,E2 10036.81} C_VEL
LIN {X 0,Y 404.621,Z 606.479,A -85,B 0,C 180,E1 10041.925,E2 10041.925} C_VEL
LIN {X 0,Y 393.627,Z 586.94,A -85,B 0,C 180,E1 10044.087,E2 10044.087} C_VEL
LIN {X 0,Y 393.725,Z 586.94,A -85,B 0,C 180,E1 10054.922,E2 10054.922} C_VEL
LIN {X 0,Y 394.202,Z 586.94,A -85,B 0,C 180,E1 10065.559,E2 10065.559} C_VEL
LIN {X 0,Y 394.998,Z 586.94,A -85,B 0,C 180,E1 10076.74,E2 10076.74} C_VEL
LIN {X 0,Y 394.796,Z 586.94,A -85,B 0,C 180,E1 10087.771,E2 10087.771} C_VEL
LIN {X 0,Y 394.222,Z 586.94,A -85,B 0,C 180,E1 10099.135,E2 10099.135} C_VEL
LIN {X 0,Y 394.087,Z 588.085,A -85,B 0,C 180,E1 10105.759,E2 10105.759} C_VEL
LIN {X 0,Y 425.397,Z 647.929,A -85,B 0,C 180,E1 10111.922,E2 10111.922} C_VEL
LIN {X 0,Y 419.19,Z 703.094,A -85,B 0,C 180,E1 10114.807,E2 10114.807} C_VEL
LIN {X 0,Y 410.588,Z 751.322,A -85,B 0,C 180,E1 10119.582,E2 10119.582} C_VEL
LIN {X 0,Y 403.173,Z 787.93,A -85,B 0,C 180,E1 10125.868,E2 10125.868} C_VEL
LIN {X 0,Y 398.374,Z 811.843,A -85,B 0,C 180,E1 10133.242,E2 10133.242} C_VEL
LIN {X 0,Y 396.887,Z 821.326,A -85,B 0,C 180,E1 10139.394,E2 10139.394} C_VEL
LIN {X 0,Y 396.44,Z 822.427,A -85,B 0,C 180,E1 10146.302,E2 10146.302} C_VEL
LIN {X 0,Y 398.358,Z 810.635,A -85,B 0,C 180,E1 10154.535,E2 10154.535} C_VEL
LIN {X 0,Y 403.005,Z 784.529,A -85,B 0,C 180,E1 10162.156,E2 10162.156} C_VEL
LIN {X 0,Y 409.736,Z 746.854,A -85,B 0,C 180,E1 10168.317,E2 10168.317} C_VEL
LIN {X 0,Y 417.131,Z 699.067,A -85,B 0,C 180,E1 10172.868,E2 10172.868} C_VEL
LIN {X 0,Y 421.751,Z 641.347,A -85,B 0,C 180,E1 10175.787,E2 10175.787} C_VEL
LIN {X 0,Y 394.694,Z 586.94,A -85,B 0,C 180,E1 10180.59,E2 10180.59} C_VEL
LIN {X 0,Y 394.229,Z 586.94,A -85,B 0,C 180,E1 10191.451,E2 10191.451} C_VEL
LIN {X 0,Y 393.785,Z 586.94,A -85,B 0,C 180,E1 10201.35,E2 10201.35} C_VEL
LIN {X 0,Y 393.604,Z 586.94,A -85,B 0,C 180,E1 10212.432,E2 10212.432} C_VEL
LIN {X 0,Y 393.533,Z 586.94,A -85,B 0,C 180,E1 10223.259,E2 10223.259} C_VEL
LIN {X 0,Y 393.838,Z 586.94,A -85,B 0,C 180,E1 10233.662,E2 10233.662} C_VEL
LIN {X 0,Y 394.742,Z 586.94,A -85,B 0,C 180,E1 10245.492,E2 10245.492} C_VEL
LIN {X 0,Y 394.927,Z 586.94,A -85,B 0,C 180,E1 10256.655,E2 10256.655} C_VEL
LIN {X 0,Y 394.828,Z 586.94,A -85,B 0,C 180,E1 10265.47,E2 10265.47} C_VEL
LIN {X 0,Y 394.387,Z 586.94,A -85,B 0,C 180,E1 10276.722,E2 10276.722} C_VEL
LIN {X 0,Y 393.968,Z 586.94,A -85,B 0,C 180,E1 10286.235,E2 10286.235} C_VEL
LIN {X 0,Y 393.889,Z 588.798,A -85,B 0,C 180,E1 10295.977,E2 10295.977} C_VEL
LIN {X 0,Y 432.83,Z 660.159,A -85,B 0,C 180,E1 10302.545,E2 10302.545} C_VEL
LIN {X 0,Y 436.411,Z 674.413,A -85,B 0,C 180,E1 10303.372,E2 10303.372} C_VEL
LIN {X 0,Y 429.653,Z 737.552,A -85,B 0,C 180,E1 10305.974,E2 10305.974} C_VEL
LIN {X 0,Y 419.17,Z 799.743,A -85,B 0,C 180,E1 10310.686,E2 10310.686} C_VEL
LIN {X 0,Y 408.095,Z 856.195,A -85,B 0,C 180,E1 10317.734,E2 10317.734} C_VEL
LIN {X 0,Y 400.119,Z 898.928,A -85,B 0,C 180,E1 10326.101,E2 10326.101} C_VEL
LIN {X 0,Y 396.241,Z 927.604,A -85,B 0,C 180,E1 10335.017,E2 10335.017} C_VEL
LIN {X 0,Y 396.046,Z 928.889,A -85,B 0,C 180,E1 10335.587,E2 10335.587} C_VEL
LIN {X 0,Y 387.515,Z 937.391,A -85,B 0,C 180,E1 10340.498,E2 10340.498} C_VEL
LIN {X 0,Y 386.903,Z 944.163,A -85,B 0,C 180,E1 10348.875,E2 10348.875} C_VEL
LIN {X 0,Y 387.212,Z 940.829,A -85,B 0,C 180,E1 10356.751,E2 10356.751} C_VEL
LIN {X 0,Y 388.815,Z 924.792,A -85,B 0,C 180,E1 10365.854,E2 10365.854} C_VEL
LIN {X 0,Y 393.479,Z 892.024,A -85,B 0,C 180,E1 10375.603,E2 10375.603} C_VEL
LIN {X 0,Y 402.634,Z 844.517,A -85,B 0,C 180,E1 10384.26,E2 10384.26} C_VEL
LIN {X 0,Y 413.928,Z 787.164,A -85,B 0,C 180,E1 10390.859,E2 10390.859} C_VEL
LIN {X 0,Y 423.814,Z 723.793,A -85,B 0,C 180,E1 10395.262,E2 10395.262} C_VEL
LIN {X 0,Y 428.119,Z 668.506,A -85,B 0,C 180,E1 10397.445,E2 10397.445} C_VEL
LIN {X 0,Y 399.32,Z 610.333,A -85,B 0,C 180,E1 10402.622,E2 10402.622} C_VEL
LIN {X 0,Y 385.582,Z 586.94,A -85,B 0,C 180,E1 10405.604,E2 10405.604} C_VEL
LIN {X 0,Y 385.727,Z 586.94,A -85,B 0,C 180,E1 10415.659,E2 10415.659} C_VEL
LIN {X 0,Y 386.286,Z 586.94,A -85,B 0,C 180,E1 10427.571,E2 10427.571} C_VEL
LIN {X 0,Y 387.401,Z 586.94,A -85,B 0,C 180,E1 10438.921,E2 10438.921} C_VEL
LIN {X 0,Y 386.624,Z 586.94,A -85,B 0,C 180,E1 10450.213,E2 10450.213} C_VEL
LIN {X 0,Y 386.196,Z 586.94,A -85,B 0,C 180,E1 10459.549,E2 10459.549} C_VEL
LIN {X 0,Y 386.069,Z 588.181,A -85,B 0,C 180,E1 10464.413,E2 10464.413} C_VEL
LIN {X 0,Y 417.551,Z 646.899,A -85,B 0,C 180,E1 10470.938,E2 10470.938} C_VEL
LIN {X 0,Y 417.82,Z 665.033,A -85,B 0,C 180,E1 10471.879,E2 10471.879} C_VEL
LIN {X 0,Y 410.175,Z 719.275,A -85,B 0,C 180,E1 10475.415,E2 10475.415} C_VEL
LIN {X 0,Y 401.357,Z 763.529,A -85,B 0,C 180,E1 10480.624,E2 10480.624} C_VEL
LIN {X 0,Y 393.868,Z 797.625,A -85,B 0,C 180,E1 10487.605,E2 10487.605} C_VEL
LIN {X 0,Y 389.909,Z 818.074,A -85,B 0,C 180,E1 10495.645,E2 10495.645} C_VEL
LIN {X 0,Y 388.358,Z 824.398,A -85,B 0,C 180,E1 10503.298,E2 10503.298} C_VEL
LIN {X 0,Y 389.516,Z 817.824,A -85,B 0,C 180,E1 10511.734,E2 10511.734} C_VEL
LIN {X 0,Y 392.74,Z 798.142,A -85,B 0,C 180,E1 10519.482,E2 10519.482} C_VEL
LIN {X 0,Y 399.26,Z 764.679,A -85,B 0,C 180,E1 10526.46,E2 10526.46} C_VEL
LIN {X 0,Y 407.651,Z 718.297,A -85,B 0,C 180,E1 10532.001,E2 10532.001} C_VEL
LIN {X 0,Y 414.869,Z 664.013,A -85,B 0,C 180,E1 10535.502,E2 10535.502} C_VEL
LIN {X 0,Y 414.764,Z 642.836,A -85,B 0,C 180,E1 10536.481,E2 10536.481} C_VEL
LIN {X 0,Y 386.619,Z 586.94,A -85,B 0,C 180,E1 10541.707,E2 10541.707} C_VEL
LIN {X 0,Y 386.104,Z 586.94,A -85,B 0,C 180,E1 10552.48,E2 10552.48} C_VEL
LIN {X 0,Y 385.659,Z 586.94,A -85,B 0,C 180,E1 10562.177,E2 10562.177} C_VEL
LIN {X 0,Y 385.578,Z 586.94,A -85,B 0,C 180,E1 10573.532,E2 10573.532} C_VEL
LIN {X 0,Y 385.522,Z 586.94,A -85,B 0,C 180,E1 10585.16,E2 10585.16} C_VEL
LIN {X 0,Y 385.78,Z 586.94,A -85,B 0,C 180,E1 10595.568,E2 10595.568} C_VEL
LIN {X 0,Y 386.742,Z 586.94,A -85,B 0,C 180,E1 10607.498,E2 10607.498} C_VEL
LIN {X 0,Y 387.044,Z 586.94,A -85,B 0,C 180,E1 10619.091,E2 10619.091} C_VEL
LIN {X 0,Y 386.723,Z 586.94,A -85,B 0,C 180,E1 10630.123,E2 10630.123} C_VEL
LIN {X 0,Y 386.086,Z 586.94,A -85,B 0,C 180,E1 10641.87,E2 10641.87} C_VEL
LIN {X 0,Y 385.576,Z 586.94,A -85,B 0,C 180,E1 10653.412,E2 10653.412} C_VEL
LIN {X 0,Y 385.904,Z 589.098,A -85,B 0,C 180,E1 10654.791,E2 10654.791} C_VEL
LIN {X 0,Y 425.513,Z 660.217,A -85,B 0,C 180,E1 10661.721,E2 10661.721} C_VEL
LIN {X 0,Y 430.083,Z 676.49,A -85,B 0,C 180,E1 10662.75,E2 10662.75} C_VEL
LIN {X 0,Y 422.899,Z 739.518,A -85,B 0,C 180,E1 10665.452,E2 10665.452} C_VEL
LIN {X 0,Y 411.853,Z 801.402,A -85,B 0,C 180,E1 10670.296,E2 10670.296} C_VEL
LIN {X 0,Y 400.616,Z 855.995,A -85,B 0,C 180,E1 10677.299,E2 10677.299} C_VEL
LIN {X 0,Y 392.128,Z 899.288,A -85,B 0,C 180,E1 10686.023,E2 10686.023} C_VEL
LIN {X 0,Y 388.166,Z 927.612,A -85,B 0,C 180,E1 10695.278,E2 10695.278} C_VEL
LIN {X 0,Y 387.515,Z 937.391,A -85,B 0,C 180,E1 10700.498,E2 10700.498} C_VEL
LIN {X 0,Y 379.263,Z 941.594,A -85,B 0,C 180,E1 10705.636,E2 10705.636} C_VEL
LIN {X 0,Y 379.426,Z 942.207,A -85,B 0,C 180,E1 10713.438,E2 10713.438} C_VEL
LIN {X 0,Y 379.806,Z 930.999,A -85,B 0,C 180,E1 10722.693,E2 10722.693} C_VEL
LIN {X 0,Y 382.575,Z 907.562,A -85,B 0,C 180,E1 10731.657,E2 10731.657} C_VEL
LIN {X 0,Y 389.593,Z 870.134,A -85,B 0,C 180,E1 10740.421,E2 10740.421} C_VEL
LIN {X 0,Y 400.573,Z 818.839,A -85,B 0,C 180,E1 10748.137,E2 10748.137} C_VEL
LIN {X 0,Y 412.44,Z 758.508,A -85,B 0,C 180,E1 10753.785,E2 10753.785} C_VEL
LIN {X 0,Y 421.148,Z 696.583,A -85,B 0,C 180,E1 10757.097,E2 10757.097} C_VEL
LIN {X 0,Y 421.673,Z 670.706,A -85,B 0,C 180,E1 10758.122,E2 10758.122} C_VEL
LIN {X 0,Y 394.048,Z 614.53,A -85,B 0,C 180,E1 10763.339,E2 10763.339} C_VEL
LIN {X 0,Y 377.533,Z 586.94,A -85,B 0,C 180,E1 10767.203,E2 10767.203} C_VEL
LIN {X 0,Y 377.694,Z 586.94,A -85,B 0,C 180,E1 10777.618,E2 10777.618} C_VEL
LIN {X 0,Y 378.487,Z 586.94,A -85,B 0,C 180,E1 10789.654,E2 10789.654} C_VEL
LIN {X 0,Y 379.406,Z 586.94,A -85,B 0,C 180,E1 10798.898,E2 10798.898} C_VEL
LIN {X 0,Y 378.564,Z 586.94,A -85,B 0,C 180,E1 10810.859,E2 10810.859} C_VEL
LIN {X 0,Y 378.058,Z 586.94,A -85,B 0,C 180,E1 10822.454,E2 10822.454} C_VEL
LIN {X 0,Y 385.857,Z 601.214,A -85,B 0,C 180,E1 10824.814,E2 10824.814} C_VEL
LIN {X 0,Y 412.798,Z 653.486,A -85,B 0,C 180,E1 10830.655,E2 10830.655} C_VEL
LIN {X 0,Y 405.455,Z 710.018,A -85,B 0,C 180,E1 10833.9,E2 10833.9} C_VEL
LIN {X 0,Y 396.029,Z 757.043,A -85,B 0,C 180,E1 10838.947,E2 10838.947} C_VEL
LIN {X 0,Y 387.653,Z 793.191,A -85,B 0,C 180,E1 10845.718,E2 10845.718} C_VEL
LIN {X 0,Y 382.642,Z 815.753,A -85,B 0,C 180,E1 10853.387,E2 10853.387} C_VEL
LIN {X 0,Y 380.908,Z 824.512,A -85,B 0,C 180,E1 10860.134,E2 10860.134} C_VEL
LIN {X 0,Y 380.832,Z 823.957,A -85,B 0,C 180,E1 10867.757,E2 10867.757} C_VEL
LIN {X 0,Y 383.306,Z 810.611,A -85,B 0,C 180,E1 10876.008,E2 10876.008} C_VEL
LIN {X 0,Y 388.869,Z 782.368,A -85,B 0,C 180,E1 10883.897,E2 10883.897} C_VEL
LIN {X 0,Y 396.906,Z 742.293,A -85,B 0,C 180,E1 10890.171,E2 10890.171} C_VEL
LIN {X 0,Y 405.138,Z 692.01,A -85,B 0,C 180,E1 10894.679,E2 10894.679} C_VEL
LIN {X 0,Y 408.375,Z 645.792,A -85,B 0,C 180,E1 10897.082,E2 10897.082} C_VEL
LIN {X 0,Y 378.559,Z 586.94,A -85,B 0,C 180,E1 10902.738,E2 10902.738} C_VEL
LIN {X 0,Y 378.135,Z 586.94,A -85,B 0,C 180,E1 10912.412,E2 10912.412} C_VEL
LIN {X 0,Y 377.568,Z 586.94,A -85,B 0,C 180,E1 10922.861,E2 10922.861} C_VEL
LIN {X 0,Y 377.454,Z 586.94,A -85,B 0,C 180,E1 10931.906,E2 10931.906} C_VEL
LIN {X 0,Y 377.465,Z 586.94,A -85,B 0,C 180,E1 10941.626,E2 10941.626} C_VEL
LIN {X 0,Y 377.722,Z 586.94,A -85,B 0,C 180,E1 10952.445,E2 10952.445} C_VEL
LIN {X 0,Y 378.595,Z 586.94,A -85,B 0,C 180,E1 10964.859,E2 10964.859} C_VEL
LIN {X 0,Y 378.935,Z 586.94,A -85,B 0,C 180,E1 10976.514,E2 10976.514} C_VEL
LIN {X 0,Y 378.828,Z 586.94,A -85,B 0,C 180,E1 10985.701,E2 10985.701} C_VEL
LIN {X 0,Y 378.267,Z 586.94,A -85,B 0,C 180,E1 10997.457,E2 10997.457} C_VEL
LIN {X 0,Y 377.836,Z 586.94,A -85,B 0,C 180,E1 11007.447,E2 11007.447} C_VEL
LIN {X 0,Y 377.774,Z 588.662,A -85,B 0,C 180,E1 11013.491,E2 11013.491} C_VEL
LIN {X 0,Y 417.361,Z 658.908,A -85,B 0,C 180,E1 11020.722,E2 11020.722} C_VEL
LIN {X 0,Y 423.742,Z 678.823,A -85,B 0,C 180,E1 11022.137,E2 11022.137} C_VEL
LIN {X 0,Y 415.999,Z 742.221,A -85,B 0,C 180,E1 11024.954,E2 11024.954} C_VEL
LIN {X 0,Y 404.702,Z 802.229,A -85,B 0,C 180,E1 11029.808,E2 11029.808} C_VEL
LIN {X 0,Y 393.002,Z 856.37,A -85,B 0,C 180,E1 11036.946,E2 11036.946} C_VEL
LIN {X 0,Y 384.27,Z 899.109,A -85,B 0,C 180,E1 11045.812,E2 11045.812} C_VEL
LIN {X 0,Y 380.301,Z 926.362,A -85,B 0,C 180,E1 11054.966,E2 11054.966} C_VEL
LIN {X 0,Y 379.333,Z 940.655,A -85,B 0,C 180,E1 11064.259,E2 11064.259} C_VEL
LIN {X 0,Y 379.263,Z 941.594,A -85,B 0,C 180,E1 11065.636,E2 11065.636} C_VEL
LIN {X 0,Y 371.262,Z 941.75,A -85,B 0,C 180,E1 11070.931,E2 11070.931} C_VEL
LIN {X 0,Y 371.752,Z 935.555,A -85,B 0,C 180,E1 11079.396,E2 11079.396} C_VEL
LIN {X 0,Y 373.432,Z 915.75,A -85,B 0,C 180,E1 11088.97,E2 11088.97} C_VEL
LIN {X 0,Y 379.166,Z 882.861,A -85,B 0,C 180,E1 11098.125,E2 11098.125} C_VEL
LIN {X 0,Y 389.561,Z 835.821,A -85,B 0,C 180,E1 11106.444,E2 11106.444} C_VEL
LIN {X 0,Y 401.972,Z 778.881,A -85,B 0,C 180,E1 11112.813,E2 11112.813} C_VEL
LIN {X 0,Y 412.458,Z 715.615,A -85,B 0,C 180,E1 11117.031,E2 11117.031} C_VEL
LIN {X 0,Y 415.585,Z 673.663,A -85,B 0,C 180,E1 11118.762,E2 11118.762} C_VEL
LIN {X 0,Y 389.544,Z 619.759,A -85,B 0,C 180,E1 11123.938,E2 11123.938} C_VEL
LIN {X 0,Y 369.458,Z 586.94,A -85,B 0,C 180,E1 11128.739,E2 11128.739} C_VEL
LIN {X 0,Y 369.736,Z 586.94,A -85,B 0,C 180,E1 11139.638,E2 11139.638} C_VEL
LIN {X 0,Y 370.45,Z 586.94,A -85,B 0,C 180,E1 11149.427,E2 11149.427} C_VEL
LIN {X 0,Y 371.406,Z 586.94,A -85,B 0,C 180,E1 11158.875,E2 11158.875} C_VEL
LIN {X 0,Y 370.586,Z 586.94,A -85,B 0,C 180,E1 11170.66,E2 11170.66} C_VEL
LIN {X 0,Y 370.158,Z 588.507,A -85,B 0,C 180,E1 11181.376,E2 11181.376} C_VEL
LIN {X 0,Y 399.469,Z 639.599,A -85,B 0,C 180,E1 11188.23,E2 11188.23} C_VEL
LIN {X 0,Y 406.369,Z 660.628,A -85,B 0,C 180,E1 11190.192,E2 11190.192} C_VEL
LIN {X 0,Y 398.416,Z 714.944,A -85,B 0,C 180,E1 11193.559,E2 11193.559} C_VEL
LIN {X 0,Y 388.437,Z 761.125,A -85,B 0,C 180,E1 11198.812,E2 11198.812} C_VEL
LIN {X 0,Y 379.594,Z 797.053,A -85,B 0,C 180,E1 11205.96,E2 11205.96} C_VEL
LIN {X 0,Y 374.571,Z 818.619,A -85,B 0,C 180,E1 11214.025,E2 11214.025} C_VEL
LIN {X 0,Y 372.67,Z 826.702,A -85,B 0,C 180,E1 11222.078,E2 11222.078} C_VEL
LIN {X 0,Y 373.585,Z 821.724,A -85,B 0,C 180,E1 11231.038,E2 11231.038} C_VEL
LIN {X 0,Y 377.1,Z 802.463,A -85,B 0,C 180,E1 11239.568,E2 11239.568} C_VEL
LIN {X 0,Y 384.118,Z 770.177,A -85,B 0,C 180,E1 11246.887,E2 11246.887} C_VEL
LIN {X 0,Y 393.369,Z 724.729,A -85,B 0,C 180,E1 11252.765,E2 11252.765} C_VEL
LIN {X 0,Y 401.385,Z 671.632,A -85,B 0,C 180,E1 11256.539,E2 11256.539} C_VEL
LIN {X 0,Y 401.893,Z 648.422,A -85,B 0,C 180,E1 11257.712,E2 11257.712} C_VEL
LIN {X 0,Y 372.281,Z 592.021,A -85,B 0,C 180,E1 11263.472,E2 11263.472} C_VEL
LIN {X 0,Y 370.427,Z 586.94,A -85,B 0,C 180,E1 11264.23,E2 11264.23} C_VEL
LIN {X 0,Y 369.91,Z 586.94,A -85,B 0,C 180,E1 11275.516,E2 11275.516} C_VEL
LIN {X 0,Y 369.401,Z 586.94,A -85,B 0,C 180,E1 11286.723,E2 11286.723} C_VEL
LIN {X 0,Y 369.371,Z 586.94,A -85,B 0,C 180,E1 11297.282,E2 11297.282} C_VEL
LIN {X 0,Y 369.573,Z 586.94,A -85,B 0,C 180,E1 11309.08,E2 11309.08} C_VEL
LIN {X 0,Y 369.837,Z 586.94,A -85,B 0,C 180,E1 11319.548,E2 11319.548} C_VEL
LIN {X 0,Y 370.692,Z 586.94,A -85,B 0,C 180,E1 11329.343,E2 11329.343} C_VEL
LIN {X 0,Y 371.469,Z 586.94,A -85,B 0,C 180,E1 11341.125,E2 11341.125} C_VEL
LIN {X 0,Y 370.466,Z 586.94,A -85,B 0,C 180,E1 11352.969,E2 11352.969} C_VEL
LIN {X 0,Y 369.984,Z 586.94,A -85,B 0,C 180,E1 11362.874,E2 11362.874} C_VEL
LIN {X 0,Y 369.788,Z 588.937,A -85,B 0,C 180,E1 11372.169,E2 11372.169} C_VEL
LIN {X 0,Y 408.667,Z 656.411,A -85,B 0,C 180,E1 11379.584,E2 11379.584} C_VEL
LIN {X 0,Y 417.431,Z 680.848,A -85,B 0,C 180,E1 11381.492,E2 11381.492} C_VEL
LIN {X 0,Y 409.201,Z 744.435,A -85,B 0,C 180,E1 11384.418,E2 11384.418} C_VEL
LIN {X 0,Y 396.822,Z 806.565,A -85,B 0,C 180,E1 11389.676,E2 11389.676} C_VEL
LIN {X 0,Y 384.624,Z 860.022,A -85,B 0,C 180,E1 11397.145,E2 11397.145} C_VEL
LIN {X 0,Y 375.922,Z 900.975,A -85,B 0,C 180,E1 11406.191,E2 11406.191} C_VEL
LIN {X 0,Y 372.231,Z 926.371,A -85,B 0,C 180,E1 11415.237,E2 11415.237} C_VEL
LIN {X 0,Y 371.401,Z 939.436,A -85,B 0,C 180,E1 11424.136,E2 11424.136} C_VEL
LIN {X 0,Y 371.262,Z 941.75,A -85,B 0,C 180,E1 11430.931,E2 11430.931} C_VEL
LIN {X 0,Y 363.416,Z 937.832,A -85,B 0,C 180,E1 11436.313,E2 11436.313} C_VEL
LIN {X 0,Y 364.934,Z 922.523,A -85,B 0,C 180,E1 11446.16,E2 11446.16} C_VEL
LIN {X 0,Y 369.877,Z 891.333,A -85,B 0,C 180,E1 11456.337,E2 11456.337} C_VEL
LIN {X 0,Y 379.618,Z 847.624,A -85,B 0,C 180,E1 11465.147,E2 11465.147} C_VEL
LIN {X 0,Y 392.122,Z 793.359,A -85,B 0,C 180,E1 11472.115,E2 11472.115} C_VEL
LIN {X 0,Y 404.181,Z 729.118,A -85,B 0,C 180,E1 11477.064,E2 11477.064} C_VEL
LIN {X 0,Y 409.537,Z 676.659,A -85,B 0,C 180,E1 11479.403,E2 11479.403} C_VEL
LIN {X 0,Y 384.639,Z 624.159,A -85,B 0,C 180,E1 11484.655,E2 11484.655} C_VEL
LIN {X 0,Y 361.457,Z 586.94,A -85,B 0,C 180,E1 11490.769,E2 11490.769} C_VEL
LIN {X 0,Y 361.834,Z 586.94,A -85,B 0,C 180,E1 11501.722,E2 11501.722} C_VEL
LIN {X 0,Y 362.593,Z 586.94,A -85,B 0,C 180,E1 11511.627,E2 11511.627} C_VEL
LIN {X 0,Y 363.009,Z 586.94,A -85,B 0,C 180,E1 11521.243,E2 11521.243} C_VEL
LIN {X 0,Y 362.55,Z 586.94,A -85,B 0,C 180,E1 11530.899,E2 11530.899} C_VEL
LIN {X 0,Y 362.282,Z 588.905,A -85,B 0,C 180,E1 11539.646,E2 11539.646} C_VEL
LIN {X 0,Y 390.195,Z 635.608,A -85,B 0,C 180,E1 11546.681,E2 11546.681} C_VEL
LIN {X 0,Y 400.304,Z 662.577,A -85,B 0,C 180,E1 11549.49,E2 11549.49} C_VEL
LIN {X 0,Y 391.748,Z 717.687,A -85,B 0,C 180,E1 11553.011,E2 11553.011} C_VEL
LIN {X 0,Y 381.092,Z 764.074,A -85,B 0,C 180,E1 11558.495,E2 11558.495} C_VEL
LIN {X 0,Y 371.783,Z 799.688,A -85,B 0,C 180,E1 11565.921,E2 11565.921} C_VEL
LIN {X 0,Y 366.799,Z 819.96,A -85,B 0,C 180,E1 11573.825,E2 11573.825} C_VEL
LIN {X 0,Y 364.839,Z 827.739,A -85,B 0,C 180,E1 11581.425,E2 11581.425} C_VEL
LIN {X 0,Y 365.596,Z 823.724,A -85,B 0,C 180,E1 11590.607,E2 11590.607} C_VEL
LIN {X 0,Y 369.115,Z 805.427,A -85,B 0,C 180,E1 11599.34,E2 11599.34} C_VEL
LIN {X 0,Y 376.516,Z 772.825,A -85,B 0,C 180,E1 11607.113,E2 11607.113} C_VEL
LIN {X 0,Y 386.138,Z 728.485,A -85,B 0,C 180,E1 11613.099,E2 11613.099} C_VEL
LIN {X 0,Y 394.726,Z 674.872,A -85,B 0,C 180,E1 11617.109,E2 11617.109} C_VEL
LIN {X 0,Y 395.505,Z 651.354,A -85,B 0,C 180,E1 11618.343,E2 11618.343} C_VEL
LIN {X 0,Y 367.708,Z 597.591,A -85,B 0,C 180,E1 11624.014,E2 11624.014} C_VEL
LIN {X 0,Y 362.428,Z 586.94,A -85,B 0,C 180,E1 11625.4,E2 11625.4} C_VEL
LIN {X 0,Y 361.81,Z 586.94,A -85,B 0,C 180,E1 11636.13,E2 11636.13} C_VEL
LIN {X 0,Y 361.314,Z 586.94,A -85,B 0,C 180,E1 11647.519,E2 11647.519} C_VEL
LIN {X 0,Y 361.346,Z 586.94,A -85,B 0,C 180,E1 11659.347,E2 11659.347} C_VEL
LIN {X 0,Y 361.552,Z 586.94,A -85,B 0,C 180,E1 11671.099,E2 11671.099} C_VEL
LIN {X 0,Y 362.044,Z 586.94,A -85,B 0,C 180,E1 11681.637,E2 11681.637} C_VEL
LIN {X 0,Y 362.799,Z 586.94,A -85,B 0,C 180,E1 11691.539,E2 11691.539} C_VEL
LIN {X 0,Y 363.452,Z 586.94,A -85,B 0,C 180,E1 11701.15,E2 11701.15} C_VEL
LIN {X 0,Y 362.417,Z 586.94,A -85,B 0,C 180,E1 11713.262,E2 11713.262} C_VEL
LIN {X 0,Y 361.904,Z 586.94,A -85,B 0,C 180,E1 11723.415,E2 11723.415} C_VEL
LIN {X 0,Y 361.75,Z 588.543,A -85,B 0,C 180,E1 11730.731,E2 11730.731} C_VEL
LIN {X 0,Y 401.2,Z 656.506,A -85,B 0,C 180,E1 11738.613,E2 11738.613} C_VEL
LIN {X 0,Y 411.156,Z 682.812,A -85,B 0,C 180,E1 11740.831,E2 11740.831} C_VEL
LIN {X 0,Y 402.696,Z 745.032,A -85,B 0,C 180,E1 11743.766,E2 11743.766} C_VEL
LIN {X 0,Y 389.7,Z 807.383,A -85,B 0,C 180,E1 11749.161,E2 11749.161} C_VEL
LIN {X 0,Y 377.002,Z 860.383,A -85,B 0,C 180,E1 11756.778,E2 11756.778} C_VEL
LIN {X 0,Y 368.047,Z 900.686,A -85,B 0,C 180,E1 11765.972,E2 11765.972} C_VEL
LIN {X 0,Y 364.187,Z 926.383,A -85,B 0,C 180,E1 11775.521,E2 11775.521} C_VEL
LIN {X 0,Y 363.467,Z 938.221,A -85,B 0,C 180,E1 11784.008,E2 11784.008} C_VEL
LIN {X 0,Y 363.554,Z 939.744,A -85,B 0,C 180,E1 11793.589,E2 11793.589} C_VEL
LIN {X 0,Y 363.416,Z 937.832,A -85,B 0,C 180,E1 11796.313,E2 11796.313} C_VEL
LIN {X 0,Y 355.862,Z 930.202,A -85,B 0,C 180,E1 11801.739,E2 11801.739} C_VEL
LIN {X 0,Y 358.274,Z 909.528,A -85,B 0,C 180,E1 11811.101,E2 11811.101} C_VEL
LIN {X 0,Y 365.656,Z 873.662,A -85,B 0,C 180,E1 11820.747,E2 11820.747} C_VEL
LIN {X 0,Y 377.778,Z 824.756,A -85,B 0,C 180,E1 11829.061,E2 11829.061} C_VEL
LIN {X 0,Y 391.12,Z 767.541,A -85,B 0,C 180,E1 11835.127,E2 11835.127} C_VEL
LIN {X 0,Y 401.877,Z 705.195,A -85,B 0,C 180,E1 11838.947,E2 11838.947} C_VEL
LIN {X 0,Y 403.145,Z 678.638,A -85,B 0,C 180,E1 11840.156,E2 11840.156} C_VEL
LIN {X 0,Y 379.428,Z 627.86,A -85,B 0,C 180,E1 11845.476,E2 11845.476} C_VEL
LIN {X 0,Y 353.427,Z 586.94,A -85,B 0,C 180,E1 11852.518,E2 11852.518} C_VEL
LIN {X 0,Y 354.023,Z 586.94,A -85,B 0,C 180,E1 11864.675,E2 11864.675} C_VEL
LIN {X 0,Y 354.923,Z 586.94,A -85,B 0,C 180,E1 11876.371,E2 11876.371} C_VEL
LIN {X 0,Y 354.817,Z 586.94,A -85,B 0,C 180,E1 11886.183,E2 11886.183} C_VEL
LIN {X 0,Y 354.3,Z 588.621,A -85,B 0,C 180,E1 11897.65,E2 11897.65} C_VEL
LIN {X 0,Y 381.357,Z 632.646,A -85,B 0,C 180,E1 11905.11,E2 11905.11} C_VEL
LIN {X 0,Y 394.216,Z 665.385,A -85,B 0,C 180,E1 11908.798,E2 11908.798} C_VEL
LIN {X 0,Y 385.105,Z 720.252,A -85,B 0,C 180,E1 11912.438,E2 11912.438} C_VEL
LIN {X 0,Y 374.074,Z 765.893,A -85,B 0,C 180,E1 11917.989,E2 11917.989} C_VEL
LIN {X 0,Y 364.272,Z 801.263,A -85,B 0,C 180,E1 11925.569,E2 11925.569} C_VEL
LIN {X 0,Y 358.873,Z 822.167,A -85,B 0,C 180,E1 11934.128,E2 11934.128} C_VEL
LIN {X 0,Y 356.782,Z 829.344,A -85,B 0,C 180,E1 11943.475,E2 11943.475} C_VEL
LIN {X 0,Y 358.197,Z 822.55,A -85,B 0,C 180,E1 11952.488,E2 11952.488} C_VEL
LIN {X 0,Y 362.707,Z 801.565,A -85,B 0,C 180,E1 11961.271,E2 11961.271} C_VEL
LIN {X 0,Y 371.081,Z 766.938,A -85,B 0,C 180,E1 11968.829,E2 11968.829} C_VEL
LIN {X 0,Y 381.18,Z 720.089,A -85,B 0,C 180,E1 11974.66,E2 11974.66} C_VEL
LIN {X 0,Y 389.768,Z 665.029,A -85,B 0,C 180,E1 11978.331,E2 11978.331} C_VEL
LIN {X 0,Y 388.244,Z 652.219,A -85,B 0,C 180,E1 11979.211,E2 11979.211} C_VEL
LIN {X 0,Y 360.6,Z 598.714,A -85,B 0,C 180,E1 11985.132,E2 11985.132} C_VEL
LIN {X 0,Y 354.267,Z 586.94,A -85,B 0,C 180,E1 11986.743,E2 11986.743} C_VEL
LIN {X 0,Y 353.641,Z 586.94,A -85,B 0,C 180,E1 11998.34,E2 11998.34} C_VEL
LIN {X 0,Y 353.286,Z 586.94,A -85,B 0,C 180,E1 12008.525,E2 12008.525} C_VEL
LIN {X 0,Y 353.333,Z 586.94,A -85,B 0,C 180,E1 12018.731,E2 12018.731} C_VEL
LIN {X 0,Y 353.52,Z 586.94,A -85,B 0,C 180,E1 12030.378,E2 12030.378} C_VEL
LIN {X 0,Y 353.96,Z 586.94,A -85,B 0,C 180,E1 12041.202,E2 12041.202} C_VEL
LIN {X 0,Y 354.768,Z 586.94,A -85,B 0,C 180,E1 12051.346,E2 12051.346} C_VEL
LIN {X 0,Y 355.454,Z 586.94,A -85,B 0,C 180,E1 12061.176,E2 12061.176} C_VEL
LIN {X 0,Y 354.367,Z 586.94,A -85,B 0,C 180,E1 12073.569,E2 12073.569} C_VEL
LIN {X 0,Y 353.874,Z 586.94,A -85,B 0,C 180,E1 12083.979,E2 12083.979} C_VEL
LIN {X 0,Y 353.825,Z 588.894,A -85,B 0,C 180,E1 12089.253,E2 12089.253} C_VEL
LIN {X 0,Y 391.983,Z 653.266,A -85,B 0,C 180,E1 12097.268,E2 12097.268} C_VEL
LIN {X 0,Y 404.921,Z 684.884,A -85,B 0,C 180,E1 12100.157,E2 12100.157} C_VEL
LIN {X 0,Y 395.968,Z 746.949,A -85,B 0,C 180,E1 12103.196,E2 12103.196} C_VEL
LIN {X 0,Y 382.771,Z 807.453,A -85,B 0,C 180,E1 12108.555,E2 12108.555} C_VEL
LIN {X 0,Y 369.515,Z 860.336,A -85,B 0,C 180,E1 12116.328,E2 12116.328} C_VEL
LIN {X 0,Y 360.069,Z 900.837,A -85,B 0,C 180,E1 12125.874,E2 12125.874} C_VEL
LIN {X 0,Y 356.161,Z 926.355,A -85,B 0,C 180,E1 12135.817,E2 12135.817} C_VEL
LIN {X 0,Y 355.526,Z 937.004,A -85,B 0,C 180,E1 12143.873,E2 12143.873} C_VEL
LIN {X 0,Y 355.642,Z 938.518,A -85,B 0,C 180,E1 12153.669,E2 12153.669} C_VEL
LIN {X 0,Y 355.862,Z 930.202,A -85,B 0,C 180,E1 12161.739,E2 12161.739} C_VEL
LIN {X 0,Y 349.202,Z 919.325,A -85,B 0,C 180,E1 12167.149,E2 12167.149} C_VEL
LIN {X 0,Y 354.768,Z 887.989,A -85,B 0,C 180,E1 12177.663,E2 12177.663} C_VEL
LIN {X 0,Y 366.071,Z 842.793,A -85,B 0,C 180,E1 12186.946,E2 12186.946} C_VEL
LIN {X 0,Y 379.93,Z 788.283,A -85,B 0,C 180,E1 12193.946,E2 12193.946} C_VEL
LIN {X 0,Y 392.414,Z 726.003,A -85,B 0,C 180,E1 12198.736,E2 12198.736} C_VEL
LIN {X 0,Y 397.264,Z 681.747,A -85,B 0,C 180,E1 12200.825,E2 12200.825} C_VEL
LIN {X 0,Y 374.852,Z 632.761,A -85,B 0,C 180,E1 12206.195,E2 12206.195} C_VEL
LIN {X 0,Y 349.223,Z 593.702,A -85,B 0,C 180,E1 12213.354,E2 12213.354} C_VEL
LIN {X 0,Y 345.467,Z 586.94,A -85,B 0,C 180,E1 12215.399,E2 12215.399} C_VEL
LIN {X 0,Y 346.083,Z 586.94,A -85,B 0,C 180,E1 12226.1,E2 12226.1} C_VEL
LIN {X 0,Y 347.382,Z 586.94,A -85,B 0,C 180,E1 12238.797,E2 12238.797} C_VEL
LIN {X 0,Y 346.46,Z 586.94,A -85,B 0,C 180,E1 12251.412,E2 12251.412} C_VEL
LIN {X 0,Y 346.533,Z 588.82,A -85,B 0,C 180,E1 12255.457,E2 12255.457} C_VEL
LIN {X 0,Y 371.92,Z 628.713,A -85,B 0,C 180,E1 12263.23,E2 12263.23} C_VEL
LIN {X 0,Y 388.278,Z 667.6,A -85,B 0,C 180,E1 12268.059,E2 12268.059} C_VEL
LIN {X 0,Y 378.763,Z 721.85,A -85,B 0,C 180,E1 12271.754,E2 12271.754} C_VEL
LIN {X 0,Y 366.914,Z 768.346,A -85,B 0,C 180,E1 12277.557,E2 12277.557} C_VEL
LIN {X 0,Y 356.61,Z 803.509,A -85,B 0,C 180,E1 12285.402,E2 12285.402} C_VEL
LIN {X 0,Y 350.947,Z 824.007,A -85,B 0,C 180,E1 12294.287,E2 12294.287} C_VEL
LIN {X 0,Y 348.894,Z 830.561,A -85,B 0,C 180,E1 12303.141,E2 12303.141} C_VEL
LIN {X 0,Y 350.204,Z 824.612,A -85,B 0,C 180,E1 12312.074,E2 12312.074} C_VEL
LIN {X 0,Y 354.655,Z 804.63,A -85,B 0,C 180,E1 12321.071,E2 12321.071} C_VEL
LIN {X 0,Y 363.115,Z 771.514,A -85,B 0,C 180,E1 12328.804,E2 12328.804} C_VEL
LIN {X 0,Y 373.824,Z 725.081,A -85,B 0,C 180,E1 12334.95,E2 12334.95} C_VEL
LIN {X 0,Y 383.015,Z 670.352,A -85,B 0,C 180,E1 12338.854,E2 12338.854} C_VEL
LIN {X 0,Y 382.514,Z 656.441,A -85,B 0,C 180,E1 12339.75,E2 12339.75} C_VEL
LIN {X 0,Y 356.443,Z 604.812,A -85,B 0,C 180,E1 12345.637,E2 12345.637} C_VEL
LIN {X 0,Y 346.172,Z 586.94,A -85,B 0,C 180,E1 12348.532,E2 12348.532} C_VEL
LIN {X 0,Y 345.468,Z 586.94,A -85,B 0,C 180,E1 12360.343,E2 12360.343} C_VEL
LIN {X 0,Y 345.227,Z 586.94,A -85,B 0,C 180,E1 12369.666,E2 12369.666} C_VEL
LIN {X 0,Y 345.216,Z 586.94,A -85,B 0,C 180,E1 12380.358,E2 12380.358} C_VEL
LIN {X 0,Y 345.501,Z 586.94,A -85,B 0,C 180,E1 12392.494,E2 12392.494} C_VEL
LIN {X 0,Y 346.213,Z 586.94,A -85,B 0,C 180,E1 12403.404,E2 12403.404} C_VEL
LIN {X 0,Y 346.864,Z 586.94,A -85,B 0,C 180,E1 12413.675,E2 12413.675} C_VEL
LIN {X 0,Y 346.974,Z 586.94,A -85,B 0,C 180,E1 12423.712,E2 12423.712} C_VEL
LIN {X 0,Y 346.341,Z 586.94,A -85,B 0,C 180,E1 12433.89,E2 12433.89} C_VEL
LIN {X 0,Y 345.648,Z 586.94,A -85,B 0,C 180,E1 12445.836,E2 12445.836} C_VEL
LIN {X 0,Y 345.919,Z 589.161,A -85,B 0,C 180,E1 12447.679,E2 12447.679} C_VEL
LIN {X 0,Y 383.414,Z 651.197,A -85,B 0,C 180,E1 12455.968,E2 12455.968} C_VEL
LIN {X 0,Y 398.739,Z 687.168,A -85,B 0,C 180,E1 12459.472,E2 12459.472} C_VEL
LIN {X 0,Y 389.116,Z 749.623,A -85,B 0,C 180,E1 12462.666,E2 12462.666} C_VEL
LIN {X 0,Y 375.356,Z 809.387,A -85,B 0,C 180,E1 12468.157,E2 12468.157} C_VEL
LIN {X 0,Y 361.946,Z 860.566,A -85,B 0,C 180,E1 12475.914,E2 12475.914} C_VEL
LIN {X 0,Y 352.06,Z 901.169,A -85,B 0,C 180,E1 12485.826,E2 12485.826} C_VEL
LIN {X 0,Y 348.164,Z 926.18,A -85,B 0,C 180,E1 12496.129,E2 12496.129} C_VEL
LIN {X 0,Y 347.653,Z 937.373,A -85,B 0,C 180,E1 12506.245,E2 12506.245} C_VEL
LIN {X 0,Y 347.706,Z 937.289,A -85,B 0,C 180,E1 12513.752,E2 12513.752} C_VEL
LIN {X 0,Y 348.044,Z 926.998,A -85,B 0,C 180,E1 12523.167,E2 12523.167} C_VEL
LIN {X 0,Y 349.202,Z 919.325,A -85,B 0,C 180,E1 12527.149,E2 12527.149} C_VEL
LIN {X 0,Y 342.983,Z 905.663,A -85,B 0,C 180,E1 12532.482,E2 12532.482} C_VEL
LIN {X 0,Y 352.34,Z 866.82,A -85,B 0,C 180,E1 12542.997,E2 12542.997} C_VEL
LIN {X 0,Y 366.194,Z 815.648,A -85,B 0,C 180,E1 12551.52,E2 12551.52} C_VEL
LIN {X 0,Y 381.157,Z 754.925,A -85,B 0,C 180,E1 12557.594,E2 12557.594} C_VEL
LIN {X 0,Y 391.711,Z 693.949,A -85,B 0,C 180,E1 12560.977,E2 12560.977} C_VEL
LIN {X 0,Y 389.579,Z 679.478,A -85,B 0,C 180,E1 12562.052,E2 12562.052} C_VEL
LIN {X 0,Y 367.414,Z 632.463,A -85,B 0,C 180,E1 12567.672,E2 12567.672} C_VEL
LIN {X 0,Y 344.144,Z 598.198,A -85,B 0,C 180,E1 12574.708,E2 12574.708} C_VEL
LIN {X 0,Y 337.498,Z 586.94,A -85,B 0,C 180,E1 12577.593,E2 12577.593} C_VEL
LIN {X 0,Y 338.236,Z 586.94,A -85,B 0,C 180,E1 12588.407,E2 12588.407} C_VEL
LIN {X 0,Y 339.371,Z 586.94,A -85,B 0,C 180,E1 12598.768,E2 12598.768} C_VEL
LIN {X 0,Y 338.584,Z 586.94,A -85,B 0,C 180,E1 12609.071,E2 12609.071} C_VEL
LIN {X 0,Y 338.586,Z 588.923,A -85,B 0,C 180,E1 12612.83,E2 12612.83} C_VEL
LIN {X 0,Y 360.531,Z 622.005,A -85,B 0,C 180,E1 12620.601,E2 12620.601} C_VEL
LIN {X 0,Y 381.635,Z 666.313,A -85,B 0,C 180,E1 12626.927,E2 12626.927} C_VEL
LIN {X 0,Y 372.635,Z 722.778,A -85,B 0,C 180,E1 12630.978,E2 12630.978} C_VEL
LIN {X 0,Y 360.329,Z 768.894,A -85,B 0,C 180,E1 12636.799,E2 12636.799} C_VEL
LIN {X 0,Y 349.395,Z 804.272,A -85,B 0,C 180,E1 12644.772,E2 12644.772} C_VEL
LIN {X 0,Y 343.435,Z 824.352,A -85,B 0,C 180,E1 12653.381,E2 12653.381} C_VEL
LIN {X 0,Y 341.086,Z 831.747,A -85,B 0,C 180,E1 12662.152,E2 12662.152} C_VEL
LIN {X 0,Y 342.182,Z 826.662,A -85,B 0,C 180,E1 12671.597,E2 12671.597} C_VEL
LIN {X 0,Y 346.537,Z 807.958,A -85,B 0,C 180,E1 12680.777,E2 12680.777} C_VEL
LIN {X 0,Y 355.129,Z 775.821,A -85,B 0,C 180,E1 12688.777,E2 12688.777} C_VEL
LIN {X 0,Y 366.326,Z 730.454,A -85,B 0,C 180,E1 12695.175,E2 12695.175} C_VEL
LIN {X 0,Y 376.142,Z 676.4,A -85,B 0,C 180,E1 12699.348,E2 12699.348} C_VEL
LIN {X 0,Y 376.162,Z 659.128,A -85,B 0,C 180,E1 12700.461,E2 12700.461} C_VEL
LIN {X 0,Y 351.51,Z 609.828,A -85,B 0,C 180,E1 12706.331,E2 12706.331} C_VEL
LIN {X 0,Y 337.994,Z 586.94,A -85,B 0,C 180,E1 12709.878,E2 12709.878} C_VEL
LIN {X 0,Y 337.396,Z 586.94,A -85,B 0,C 180,E1 12721.149,E2 12721.149} C_VEL
LIN {X 0,Y 337.113,Z 586.94,A -85,B 0,C 180,E1 12731.986,E2 12731.986} C_VEL
LIN {X 0,Y 337.121,Z 586.94,A -85,B 0,C 180,E1 12742.533,E2 12742.533} C_VEL
LIN {X 0,Y 337.522,Z 586.94,A -85,B 0,C 180,E1 12754.671,E2 12754.671} C_VEL
LIN {X 0,Y 338.415,Z 586.94,A -85,B 0,C 180,E1 12765.677,E2 12765.677} C_VEL
LIN {X 0,Y 338.919,Z 586.94,A -85,B 0,C 180,E1 12776.101,E2 12776.101} C_VEL
LIN {X 0,Y 338.764,Z 586.94,A -85,B 0,C 180,E1 12786.378,E2 12786.378} C_VEL
LIN {X 0,Y 338.133,Z 586.94,A -85,B 0,C 180,E1 12796.902,E2 12796.902} C_VEL
LIN {X 0,Y 337.824,Z 588.557,A -85,B 0,C 180,E1 12805.917,E2 12805.917} C_VEL
LIN {X 0,Y 375.791,Z 650.876,A -85,B 0,C 180,E1 12814.796,E2 12814.796} C_VEL
LIN {X 0,Y 392.301,Z 690.921,A -85,B 0,C 180,E1 12818.824,E2 12818.824} C_VEL
LIN {X 0,Y 381.713,Z 754.768,A -85,B 0,C 180,E1 12822.282,E2 12822.282} C_VEL
LIN {X 0,Y 366.978,Z 814.862,A -85,B 0,C 180,E1 12828.184,E2 12828.184} C_VEL
LIN {X 0,Y 353.286,Z 864.509,A -85,B 0,C 180,E1 12836.263,E2 12836.263} C_VEL
LIN {X 0,Y 343.955,Z 901.811,A -85,B 0,C 180,E1 12845.913,E2 12845.913} C_VEL
LIN {X 0,Y 340.147,Z 926,A -85,B 0,C 180,E1 12856.453,E2 12856.453} C_VEL
LIN {X 0,Y 339.749,Z 936.157,A -85,B 0,C 180,E1 12866.157,E2 12866.157} C_VEL
LIN {X 0,Y 339.791,Z 936.059,A -85,B 0,C 180,E1 12873.84,E2 12873.84} C_VEL
LIN {X 0,Y 340.167,Z 925.594,A -85,B 0,C 180,E1 12883.544,E2 12883.544} C_VEL
LIN {X 0,Y 342.983,Z 905.663,A -85,B 0,C 180,E1 12892.482,E2 12892.482} C_VEL
LIN {X 0,Y 338.775,Z 889.442,A -85,B 0,C 180,E1 12897.773,E2 12897.773} C_VEL
LIN {X 0,Y 350.738,Z 845.868,A -85,B 0,C 180,E1 12907.549,E2 12907.549} C_VEL
LIN {X 0,Y 366.34,Z 790.264,A -85,B 0,C 180,E1 12915.2,E2 12915.2} C_VEL
LIN {X 0,Y 380.325,Z 727.233,A -85,B 0,C 180,E1 12920.28,E2 12920.28} C_VEL
LIN {X 0,Y 385.438,Z 687.352,A -85,B 0,C 180,E1 12922.291,E2 12922.291} C_VEL
LIN {X 0,Y 364.917,Z 640.435,A -85,B 0,C 180,E1 12927.96,E2 12927.96} C_VEL
LIN {X 0,Y 341.986,Z 605.695,A -85,B 0,C 180,E1 12935.078,E2 12935.078} C_VEL
LIN {X 0,Y 329.646,Z 586.94,A -85,B 0,C 180,E1 12941.475,E2 12941.475} C_VEL
LIN {X 0,Y 330.582,Z 586.94,A -85,B 0,C 180,E1 12953.463,E2 12953.463} C_VEL
LIN {X 0,Y 331.002,Z 586.94,A -85,B 0,C 180,E1 12961.363,E2 12961.363} C_VEL
LIN {X 0,Y 330.753,Z 588.923,A -85,B 0,C 180,E1 12969.625,E2 12969.625} C_VEL
LIN {X 0,Y 348.974,Z 615.103,A -85,B 0,C 180,E1 12977.435,E2 12977.435} C_VEL
LIN {X 0,Y 371.188,Z 656.75,A -85,B 0,C 180,E1 12984.491,E2 12984.491} C_VEL
LIN {X 0,Y 376.111,Z 675.501,A -85,B 0,C 180,E1 12986.683,E2 12986.683} C_VEL
LIN {X 0,Y 364.998,Z 730.279,A -85,B 0,C 180,E1 12990.814,E2 12990.814} C_VEL
LIN {X 0,Y 351.932,Z 775.529,A -85,B 0,C 180,E1 12997.089,E2 12997.089} C_VEL
LIN {X 0,Y 341.434,Z 807.535,A -85,B 0,C 180,E1 13004.897,E2 13004.897} C_VEL
LIN {X 0,Y 335.288,Z 827.006,A -85,B 0,C 180,E1 13014.112,E2 13014.112} C_VEL
LIN {X 0,Y 333.111,Z 833.024,A -85,B 0,C 180,E1 13022.73,E2 13022.73} C_VEL
LIN {X 0,Y 334.647,Z 826.506,A -85,B 0,C 180,E1 13032.858,E2 13032.858} C_VEL
LIN {X 0,Y 339.988,Z 805.66,A -85,B 0,C 180,E1 13042.306,E2 13042.306} C_VEL
LIN {X 0,Y 349.755,Z 770.867,A -85,B 0,C 180,E1 13050.461,E2 13050.461} C_VEL
LIN {X 0,Y 361.346,Z 724.2,A -85,B 0,C 180,E1 13056.633,E2 13056.633} C_VEL
LIN {X 0,Y 371.067,Z 669.852,A -85,B 0,C 180,E1 13060.503,E2 13060.503} C_VEL
LIN {X 0,Y 356.674,Z 631.957,A -85,B 0,C 180,E1 13064.688,E2 13064.688} C_VEL
LIN {X 0,Y 329.907,Z 586.94,A -85,B 0,C 180,E1 13071.594,E2 13071.594} C_VEL
LIN {X 0,Y 329.303,Z 586.94,A -85,B 0,C 180,E1 13082.004,E2 13082.004} C_VEL
LIN {X 0,Y 329.117,Z 586.94,A -85,B 0,C 180,E1 13094.334,E2 13094.334} C_VEL
LIN {X 0,Y 329.111,Z 586.94,A -85,B 0,C 180,E1 13104.759,E2 13104.759} C_VEL
LIN {X 0,Y 329.534,Z 586.94,A -85,B 0,C 180,E1 13116.912,E2 13116.912} C_VEL
LIN {X 0,Y 330.508,Z 586.94,A -85,B 0,C 180,E1 13128.029,E2 13128.029} C_VEL
LIN {X 0,Y 331.048,Z 586.94,A -85,B 0,C 180,E1 13139.211,E2 13139.211} C_VEL
LIN {X 0,Y 330.614,Z 586.94,A -85,B 0,C 180,E1 13149.294,E2 13149.294} C_VEL
LIN {X 0,Y 329.92,Z 586.94,A -85,B 0,C 180,E1 13160.118,E2 13160.118} C_VEL
LIN {X 0,Y 329.906,Z 588.894,A -85,B 0,C 180,E1 13164.112,E2 13164.112} C_VEL
LIN {X 0,Y 366.813,Z 648.063,A -85,B 0,C 180,E1 13173.26,E2 13173.26} C_VEL
LIN {X 0,Y 386.149,Z 692.672,A -85,B 0,C 180,E1 13178.095,E2 13178.095} C_VEL
LIN {X 0,Y 375.05,Z 756.477,A -85,B 0,C 180,E1 13181.655,E2 13181.655} C_VEL
LIN {X 0,Y 359.671,Z 816.367,A -85,B 0,C 180,E1 13187.721,E2 13187.721} C_VEL
LIN {X 0,Y 345.21,Z 866.577,A -85,B 0,C 180,E1 13196.242,E2 13196.242} C_VEL
LIN {X 0,Y 335.851,Z 902.357,A -85,B 0,C 180,E1 13206.004,E2 13206.004} C_VEL
LIN {X 0,Y 332.266,Z 924.75,A -85,B 0,C 180,E1 13216.125,E2 13216.125} C_VEL
LIN {X 0,Y 331.814,Z 934.939,A -85,B 0,C 180,E1 13226.065,E2 13226.065} C_VEL
LIN {X 0,Y 331.854,Z 934.828,A -85,B 0,C 180,E1 13233.932,E2 13233.932} C_VEL
LIN {X 0,Y 332.309,Z 924.306,A -85,B 0,C 180,E1 13243.87,E2 13243.87} C_VEL
LIN {X 0,Y 337.063,Z 897.522,A -85,B 0,C 180,E1 13255.321,E2 13255.321} C_VEL
LIN {X 0,Y 338.775,Z 889.442,A -85,B 0,C 180,E1 13257.773,E2 13257.773} C_VEL
LIN {X 0,Y 335.81,Z 871.075,A -85,B 0,C 180,E1 13262.911,E2 13262.911} C_VEL
LIN {X 0,Y 350.256,Z 823.13,A -85,B 0,C 180,E1 13271.844,E2 13271.844} C_VEL
LIN {X 0,Y 366.525,Z 764.872,A -85,B 0,C 180,E1 13278.399,E2 13278.399} C_VEL
LIN {X 0,Y 378.95,Z 703.744,A -85,B 0,C 180,E1 13282.271,E2 13282.271} C_VEL
LIN {X 0,Y 379.155,Z 688.914,A -85,B 0,C 180,E1 13283.187,E2 13283.187} C_VEL
LIN {X 0,Y 359.114,Z 642.619,A -85,B 0,C 180,E1 13289.158,E2 13289.158} C_VEL
LIN {X 0,Y 336.57,Z 608.182,A -85,B 0,C 180,E1 13296.827,E2 13296.827} C_VEL
LIN {X 0,Y 324.992,Z 593.372,A -85,B 0,C 180,E1 13302.918,E2 13302.918} C_VEL
LIN {X 0,Y 321.991,Z 586.94,A -85,B 0,C 180,E1 13306.429,E2 13306.429} C_VEL
LIN {X 0,Y 323.34,Z 586.94,A -85,B 0,C 180,E1 13318.707,E2 13318.707} C_VEL
LIN {X 0,Y 323.008,Z 589.047,A -85,B 0,C 180,E1 13325.357,E2 13325.357} C_VEL
LIN {X 0,Y 334.166,Z 604.486,A -85,B 0,C 180,E1 13332.087,E2 13332.087} C_VEL
LIN {X 0,Y 354.013,Z 635.496,A -85,B 0,C 180,E1 13339.669,E2 13339.669} C_VEL
LIN {X 0,Y 370.808,Z 675.229,A -85,B 0,C 180,E1 13345.738,E2 13345.738} C_VEL
LIN {X 0,Y 359.398,Z 729.572,A -85,B 0,C 180,E1 13349.82,E2 13349.82} C_VEL
LIN {X 0,Y 345.836,Z 774.77,A -85,B 0,C 180,E1 13356.029,E2 13356.029} C_VEL
LIN {X 0,Y 334.157,Z 808.636,A -85,B 0,C 180,E1 13364.327,E2 13364.327} C_VEL
LIN {X 0,Y 327.902,Z 827.119,A -85,B 0,C 180,E1 13372.939,E2 13372.939} C_VEL
LIN {X 0,Y 325.5,Z 833.854,A -85,B 0,C 180,E1 13380.692,E2 13380.692} C_VEL
LIN {X 0,Y 326.235,Z 830.175,A -85,B 0,C 180,E1 13391,E2 13391} C_VEL
LIN {X 0,Y 330.791,Z 812.507,A -85,B 0,C 180,E1 13400.762,E2 13400.762} C_VEL
LIN {X 0,Y 339.954,Z 781.541,A -85,B 0,C 180,E1 13409.27,E2 13409.27} C_VEL
LIN {X 0,Y 352.108,Z 737.345,A -85,B 0,C 180,E1 13416.058,E2 13416.058} C_VEL
LIN {X 0,Y 362.909,Z 684.49,A -85,B 0,C 180,E1 13420.559,E2 13420.559} C_VEL
LIN {X 0,Y 363.902,Z 665.426,A -85,B 0,C 180,E1 13421.834,E2 13421.834} C_VEL
LIN {X 0,Y 341.919,Z 619.681,A -85,B 0,C 180,E1 13427.753,E2 13427.753} C_VEL
LIN {X 0,Y 321.72,Z 586.94,A -85,B 0,C 180,E1 13433.638,E2 13433.638} C_VEL
LIN {X 0,Y 321.105,Z 586.94,A -85,B 0,C 180,E1 13446.211,E2 13446.211} C_VEL
LIN {X 0,Y 321.054,Z 586.94,A -85,B 0,C 180,E1 13457.109,E2 13457.109} C_VEL
LIN {X 0,Y 321.113,Z 586.94,A -85,B 0,C 180,E1 13467.033,E2 13467.033} C_VEL
LIN {X 0,Y 321.608,Z 586.94,A -85,B 0,C 180,E1 13479.228,E2 13479.228} C_VEL
LIN {X 0,Y 322.66,Z 586.94,A -85,B 0,C 180,E1 13490.477,E2 13490.477} C_VEL
LIN {X 0,Y 323.39,Z 586.94,A -85,B 0,C 180,E1 13501.293,E2 13501.293} C_VEL
LIN {X 0,Y 322.343,Z 586.94,A -85,B 0,C 180,E1 13512.173,E2 13512.173} C_VEL
LIN {X 0,Y 321.983,Z 588.821,A -85,B 0,C 180,E1 13522.141,E2 13522.141} C_VEL
LIN {X 0,Y 358.277,Z 646.12,A -85,B 0,C 180,E1 13531.721,E2 13531.721} C_VEL
LIN {X 0,Y 380.173,Z 693.69,A -85,B 0,C 180,E1 13537.316,E2 13537.316} C_VEL
LIN {X 0,Y 368.67,Z 756.766,A -85,B 0,C 180,E1 13540.903,E2 13540.903} C_VEL
LIN {X 0,Y 353.103,Z 815.316,A -85,B 0,C 180,E1 13546.908,E2 13546.908} C_VEL
LIN {X 0,Y 337.62,Z 866.747,A -85,B 0,C 180,E1 13555.815,E2 13555.815} C_VEL
LIN {X 0,Y 327.736,Z 902.897,A -85,B 0,C 180,E1 13566.098,E2 13566.098} C_VEL
LIN {X 0,Y 324.247,Z 924.549,A -85,B 0,C 180,E1 13576.466,E2 13576.466} C_VEL
LIN {X 0,Y 323.881,Z 933.722,A -85,B 0,C 180,E1 13585.969,E2 13585.969} C_VEL
LIN {X 0,Y 323.917,Z 933.597,A -85,B 0,C 180,E1 13594.028,E2 13594.028} C_VEL
LIN {X 0,Y 324.464,Z 923.022,A -85,B 0,C 180,E1 13604.213,E2 13604.213} C_VEL
LIN {X 0,Y 329.471,Z 896.115,A -85,B 0,C 180,E1 13615.947,E2 13615.947} C_VEL
LIN {X 0,Y 335.81,Z 871.075,A -85,B 0,C 180,E1 13622.911,E2 13622.911} C_VEL
LIN {X 0,Y 334.798,Z 850.443,A -85,B 0,C 180,E1 13627.862,E2 13627.862} C_VEL
LIN {X 0,Y 351.191,Z 797.741,A -85,B 0,C 180,E1 13635.913,E2 13635.913} C_VEL
LIN {X 0,Y 366.655,Z 737.524,A -85,B 0,C 180,E1 13641.348,E2 13641.348} C_VEL
LIN {X 0,Y 373.772,Z 693.144,A -85,B 0,C 180,E1 13643.817,E2 13643.817} C_VEL
LIN {X 0,Y 355.236,Z 648.194,A -85,B 0,C 180,E1 13649.85,E2 13649.85} C_VEL
LIN {X 0,Y 334.041,Z 615.116,A -85,B 0,C 180,E1 13657.436,E2 13657.436} C_VEL
LIN {X 0,Y 322.692,Z 600.333,A -85,B 0,C 180,E1 13663.777,E2 13663.777} C_VEL
LIN {X 0,Y 318.459,Z 594.06,A -85,B 0,C 180,E1 13667.676,E2 13667.676} C_VEL
LIN {X 0,Y 316.384,Z 591.011,A -85,B 0,C 180,E1 13679.022,E2 13679.022} C_VEL
LIN {X 0,Y 321.681,Z 597.597,A -85,B 0,C 180,E1 13685.294,E2 13685.294} C_VEL
LIN {X 0,Y 332.939,Z 613.349,A -85,B 0,C 180,E1 13692.153,E2 13692.153} C_VEL
LIN {X 0,Y 352.343,Z 645.577,A -85,B 0,C 180,E1 13699.811,E2 13699.811} C_VEL
LIN {X 0,Y 364.643,Z 680.663,A -85,B 0,C 180,E1 13705.07,E2 13705.07} C_VEL
LIN {X 0,Y 352.501,Z 734.136,A -85,B 0,C 180,E1 13709.341,E2 13709.341} C_VEL
LIN {X 0,Y 338.077,Z 779.294,A -85,B 0,C 180,E1 13715.919,E2 13715.919} C_VEL
LIN {X 0,Y 325.971,Z 812.219,A -85,B 0,C 180,E1 13724.628,E2 13724.628} C_VEL
LIN {X 0,Y 319.749,Z 829.634,A -85,B 0,C 180,E1 13733.614,E2 13733.614} C_VEL
LIN {X 0,Y 317.283,Z 835.507,A -85,B 0,C 180,E1 13742.977,E2 13742.977} C_VEL
LIN {X 0,Y 319.079,Z 828.629,A -85,B 0,C 180,E1 13753.492,E2 13753.492} C_VEL
LIN {X 0,Y 325.495,Z 806.717,A -85,B 0,C 180,E1 13763.632,E2 13763.632} C_VEL
LIN {X 0,Y 336.201,Z 771.885,A -85,B 0,C 180,E1 13771.941,E2 13771.941} C_VEL
LIN {X 0,Y 348.867,Z 724.706,A -85,B 0,C 180,E1 13778.286,E2 13778.286} C_VEL
LIN {X 0,Y 358.434,Z 670.427,A -85,B 0,C 180,E1 13782.33,E2 13782.33} C_VEL
LIN {X 0,Y 337.808,Z 625.583,A -85,B 0,C 180,E1 13788.338,E2 13788.338} C_VEL
LIN {X 0,Y 313.505,Z 586.94,A -85,B 0,C 180,E1 13795.844,E2 13795.844} C_VEL
LIN {X 0,Y 313.045,Z 586.94,A -85,B 0,C 180,E1 13807.299,E2 13807.299} C_VEL
LIN {X 0,Y 312.935,Z 586.94,A -85,B 0,C 180,E1 13819.056,E2 13819.056} C_VEL
LIN {X 0,Y 313.129,Z 586.94,A -85,B 0,C 180,E1 13829.364,E2 13829.364} C_VEL
LIN {X 0,Y 313.819,Z 586.94,A -85,B 0,C 180,E1 13841.632,E2 13841.632} C_VEL
LIN {X 0,Y 314.763,Z 586.94,A -85,B 0,C 180,E1 13853.027,E2 13853.027} C_VEL
LIN {X 0,Y 314.906,Z 586.94,A -85,B 0,C 180,E1 13864.091,E2 13864.091} C_VEL
LIN {X 0,Y 314.157,Z 586.94,A -85,B 0,C 180,E1 13875.346,E2 13875.346} C_VEL
LIN {X 0,Y 314.008,Z 588.731,A -85,B 0,C 180,E1 13879.982,E2 13879.982} C_VEL
LIN {X 0,Y 348.874,Z 642.845,A -85,B 0,C 180,E1 13889.888,E2 13889.888} C_VEL
LIN {X 0,Y 373.855,Z 695.731,A -85,B 0,C 180,E1 13896.529,E2 13896.529} C_VEL
LIN {X 0,Y 361.918,Z 759.057,A -85,B 0,C 180,E1 13900.295,E2 13900.295} C_VEL
LIN {X 0,Y 345.887,Z 816.45,A -85,B 0,C 180,E1 13906.375,E2 13906.375} C_VEL
LIN {X 0,Y 330.101,Z 866.535,A -85,B 0,C 180,E1 13915.306,E2 13915.306} C_VEL
LIN {X 0,Y 319.61,Z 903.405,A -85,B 0,C 180,E1 13926.196,E2 13926.196} C_VEL
LIN {X 0,Y 316.363,Z 923.278,A -85,B 0,C 180,E1 13936.122,E2 13936.122} C_VEL
LIN {X 0,Y 315.946,Z 932.494,A -85,B 0,C 180,E1 13945.867,E2 13945.867} C_VEL
LIN {X 0,Y 315.982,Z 932.365,A -85,B 0,C 180,E1 13954.13,E2 13954.13} C_VEL
LIN {X 0,Y 316.61,Z 921.737,A -85,B 0,C 180,E1 13964.573,E2 13964.573} C_VEL
LIN {X 0,Y 321.823,Z 894.692,A -85,B 0,C 180,E1 13976.612,E2 13976.612} C_VEL
LIN {X 0,Y 333.82,Z 853.867,A -85,B 0,C 180,E1 13987.19,E2 13987.19} C_VEL
LIN {X 0,Y 334.798,Z 850.443,A -85,B 0,C 180,E1 13987.862,E2 13987.862} C_VEL
LIN {X 0,Y 335.064,Z 827.814,A -85,B 0,C 180,E1 13992.546,E2 13992.546} C_VEL
LIN {X 0,Y 352.242,Z 772.69,A -85,B 0,C 180,E1 13999.387,E2 13999.387} C_VEL
LIN {X 0,Y 366.472,Z 712.173,A -85,B 0,C 180,E1 14003.685,E2 14003.685} C_VEL
LIN {X 0,Y 367.544,Z 694.382,A -85,B 0,C 180,E1 14004.82,E2 14004.82} C_VEL
LIN {X 0,Y 350.102,Z 651.479,A -85,B 0,C 180,E1 14010.971,E2 14010.971} C_VEL
LIN {X 0,Y 330.751,Z 620.95,A -85,B 0,C 180,E1 14018.441,E2 14018.441} C_VEL
LIN {X 0,Y 318.187,Z 602.358,A -85,B 0,C 180,E1 14026.965,E2 14026.965} C_VEL
LIN {X 0,Y 315.22,Z 598.857,A -85,B 0,C 180,E1 14038.846,E2 14038.846} C_VEL
LIN {X 0,Y 320.394,Z 605.869,A -85,B 0,C 180,E1 14045.23,E2 14045.23} C_VEL
LIN {X 0,Y 333.249,Z 624.165,A -85,B 0,C 180,E1 14052.931,E2 14052.931} C_VEL
LIN {X 0,Y 352.129,Z 660.1,A -85,B 0,C 180,E1 14060.751,E2 14060.751} C_VEL
LIN {X 0,Y 358.867,Z 684.399,A -85,B 0,C 180,E1 14064.288,E2 14064.288} C_VEL
LIN {X 0,Y 345.988,Z 737.317,A -85,B 0,C 180,E1 14068.699,E2 14068.699} C_VEL
LIN {X 0,Y 331.12,Z 781.441,A -85,B 0,C 180,E1 14075.348,E2 14075.348} C_VEL
LIN {X 0,Y 318.64,Z 813.474,A -85,B 0,C 180,E1 14084.069,E2 14084.069} C_VEL
LIN {X 0,Y 311.944,Z 831.078,A -85,B 0,C 180,E1 14093.445,E2 14093.445} C_VEL
LIN {X 0,Y 309.46,Z 836.734,A -85,B 0,C 180,E1 14102.236,E2 14102.236} C_VEL
LIN {X 0,Y 310.782,Z 831.532,A -85,B 0,C 180,E1 14112.31,E2 14112.31} C_VEL
LIN {X 0,Y 316.466,Z 812.359,A -85,B 0,C 180,E1 14122.581,E2 14122.581} C_VEL
LIN {X 0,Y 327.139,Z 779.749,A -85,B 0,C 180,E1 14131.33,E2 14131.33} C_VEL
LIN {X 0,Y 340.427,Z 734.266,A -85,B 0,C 180,E1 14138.17,E2 14138.17} C_VEL
LIN {X 0,Y 352.023,Z 680.095,A -85,B 0,C 180,E1 14142.593,E2 14142.593} C_VEL
LIN {X 0,Y 349.324,Z 664.438,A -85,B 0,C 180,E1 14144.212,E2 14144.212} C_VEL
LIN {X 0,Y 325.993,Z 618.573,A -85,B 0,C 180,E1 14151.079,E2 14151.079} C_VEL
LIN {X 0,Y 305.318,Z 586.94,A -85,B 0,C 180,E1 14158.177,E2 14158.177} C_VEL
LIN {X 0,Y 304.837,Z 586.94,A -85,B 0,C 180,E1 14169.443,E2 14169.443} C_VEL
LIN {X 0,Y 304.861,Z 586.94,A -85,B 0,C 180,E1 14181.47,E2 14181.47} C_VEL
LIN {X 0,Y 305.156,Z 586.94,A -85,B 0,C 180,E1 14191.759,E2 14191.759} C_VEL
LIN {X 0,Y 306.183,Z 586.94,A -85,B 0,C 180,E1 14205.126,E2 14205.126} C_VEL
LIN {X 0,Y 306.859,Z 586.94,A -85,B 0,C 180,E1 14215.693,E2 14215.693} C_VEL
LIN {X 0,Y 306.887,Z 586.94,A -85,B 0,C 180,E1 14224.198,E2 14224.198} C_VEL
LIN {X 0,Y 306.097,Z 586.94,A -85,B 0,C 180,E1 14235.76,E2 14235.76} C_VEL
LIN {X 0,Y 306.221,Z 589.12,A -85,B 0,C 180,E1 14237.699,E2 14237.699} C_VEL
LIN {X 0,Y 338.593,Z 638.143,A -85,B 0,C 180,E1 14247.685,E2 14247.685} C_VEL
LIN {X 0,Y 364.942,Z 690.953,A -85,B 0,C 180,E1 14254.874,E2 14254.874} C_VEL
LIN {X 0,Y 367.17,Z 702.853,A -85,B 0,C 180,E1 14255.985,E2 14255.985} C_VEL
LIN {X 0,Y 353.755,Z 767.129,A -85,B 0,C 180,E1 14260.16,E2 14260.16} C_VEL
LIN {X 0,Y 336.523,Z 824.148,A -85,B 0,C 180,E1 14266.773,E2 14266.773} C_VEL
LIN {X 0,Y 320.642,Z 872.266,A -85,B 0,C 180,E1 14276.228,E2 14276.228} C_VEL
LIN {X 0,Y 311.056,Z 905.438,A -85,B 0,C 180,E1 14286.993,E2 14286.993} C_VEL
LIN {X 0,Y 308.243,Z 925.11,A -85,B 0,C 180,E1 14298.133,E2 14298.133} C_VEL
LIN {X 0,Y 307.883,Z 932.03,A -85,B 0,C 180,E1 14308.587,E2 14308.587} C_VEL
LIN {X 0,Y 308.141,Z 928.337,A -85,B 0,C 180,E1 14318.495,E2 14318.495} C_VEL
LIN {X 0,Y 309.591,Z 912.803,A -85,B 0,C 180,E1 14329.32,E2 14329.32} C_VEL
LIN {X 0,Y 316.863,Z 882.788,A -85,B 0,C 180,E1 14340.641,E2 14340.641} C_VEL
LIN {X 0,Y 331.19,Z 839.29,A -85,B 0,C 180,E1 14350.605,E2 14350.605} C_VEL
LIN {X 0,Y 335.064,Z 827.814,A -85,B 0,C 180,E1 14352.546,E2 14352.546} C_VEL
LIN {X 0,Y 336.677,Z 803.102,A -85,B 0,C 180,E1 14356.895,E2 14356.895} C_VEL
LIN {X 0,Y 353.806,Z 743.882,A -85,B 0,C 180,E1 14362.719,E2 14362.719} C_VEL
LIN {X 0,Y 362.37,Z 698.959,A -85,B 0,C 180,E1 14365.453,E2 14365.453} C_VEL
LIN {X 0,Y 345.774,Z 655.805,A -85,B 0,C 180,E1 14371.916,E2 14371.916} C_VEL
LIN {X 0,Y 326.206,Z 623.94,A -85,B 0,C 180,E1 14380.263,E2 14380.263} C_VEL
LIN {X 0,Y 315.653,Z 609.483,A -85,B 0,C 180,E1 14388.62,E2 14388.62} C_VEL
LIN {X 0,Y 314.203,Z 607.089,A -85,B 0,C 180,E1 14399.015,E2 14399.015} C_VEL
LIN {X 0,Y 319.353,Z 614.352,A -85,B 0,C 180,E1 14405.354,E2 14405.354} C_VEL
LIN {X 0,Y 333.314,Z 635.29,A -85,B 0,C 180,E1 14413.623,E2 14413.623} C_VEL
LIN {X 0,Y 350.256,Z 672.687,A -85,B 0,C 180,E1 14421.357,E2 14421.357} C_VEL
LIN {X 0,Y 353.223,Z 687.482,A -85,B 0,C 180,E1 14423.451,E2 14423.451} C_VEL
LIN {X 0,Y 339.252,Z 741.521,A -85,B 0,C 180,E1 14428.144,E2 14428.144} C_VEL
LIN {X 0,Y 323.898,Z 784.356,A -85,B 0,C 180,E1 14434.927,E2 14434.927} C_VEL
LIN {X 0,Y 310.628,Z 816.698,A -85,B 0,C 180,E1 14444.242,E2 14444.242} C_VEL
LIN {X 0,Y 303.501,Z 834.198,A -85,B 0,C 180,E1 14454.902,E2 14454.902} C_VEL
LIN {X 0,Y 301.419,Z 837.828,A -85,B 0,C 180,E1 14464.665,E2 14464.665} C_VEL
LIN {X 0,Y 304.068,Z 829.096,A -85,B 0,C 180,E1 14475.347,E2 14475.347} C_VEL
LIN {X 0,Y 311.63,Z 806.467,A -85,B 0,C 180,E1 14485.463,E2 14485.463} C_VEL
LIN {X 0,Y 323.819,Z 770.191,A -85,B 0,C 180,E1 14494.032,E2 14494.032} C_VEL
LIN {X 0,Y 337.476,Z 722.063,A -85,B 0,C 180,E1 14500.363,E2 14500.363} C_VEL
LIN {X 0,Y 345.934,Z 675.446,A -85,B 0,C 180,E1 14503.963,E2 14503.963} C_VEL
LIN {X 0,Y 325.902,Z 630.953,A -85,B 0,C 180,E1 14510.594,E2 14510.594} C_VEL
LIN {X 0,Y 299.541,Z 592.537,A -85,B 0,C 180,E1 14519.261,E2 14519.261} C_VEL
LIN {X 0,Y 297.166,Z 586.94,A -85,B 0,C 180,E1 14520.343,E2 14520.343} C_VEL
LIN {X 0,Y 296.818,Z 586.94,A -85,B 0,C 180,E1 14533.648,E2 14533.648} C_VEL
LIN {X 0,Y 296.822,Z 586.94,A -85,B 0,C 180,E1 14543.936,E2 14543.936} C_VEL
LIN {X 0,Y 297.188,Z 586.94,A -85,B 0,C 180,E1 14554.225,E2 14554.225} C_VEL
LIN {X 0,Y 298.302,Z 586.94,A -85,B 0,C 180,E1 14566.715,E2 14566.715} C_VEL
LIN {X 0,Y 299.013,Z 586.94,A -85,B 0,C 180,E1 14579.271,E2 14579.271} C_VEL
LIN {X 0,Y 298.452,Z 586.94,A -85,B 0,C 180,E1 14590.19,E2 14590.19} C_VEL
LIN {X 0,Y 298.331,Z 588.694,A -85,B 0,C 180,E1 14595.121,E2 14595.121} C_VEL
LIN {X 0,Y 330.65,Z 637.21,A -85,B 0,C 180,E1 14605.929,E2 14605.929} C_VEL
LIN {X 0,Y 356.783,Z 688.652,A -85,B 0,C 180,E1 14613.406,E2 14613.406} C_VEL
LIN {X 0,Y 360.94,Z 705.668,A -85,B 0,C 180,E1 14615.233,E2 14615.233} C_VEL
LIN {X 0,Y 347.308,Z 767.898,A -85,B 0,C 180,E1 14619.402,E2 14619.402} C_VEL
LIN {X 0,Y 329.474,Z 824.596,A -85,B 0,C 180,E1 14626.122,E2 14626.122} C_VEL
LIN {X 0,Y 313.116,Z 872.08,A -85,B 0,C 180,E1 14635.715,E2 14635.715} C_VEL
LIN {X 0,Y 302.956,Z 905.843,A -85,B 0,C 180,E1 14647.158,E2 14647.158} C_VEL
LIN {X 0,Y 300.299,Z 924.459,A -85,B 0,C 180,E1 14658.337,E2 14658.337} C_VEL
LIN {X 0,Y 299.971,Z 930.81,A -85,B 0,C 180,E1 14668.549,E2 14668.549} C_VEL
LIN {X 0,Y 300.205,Z 927.091,A -85,B 0,C 180,E1 14678.721,E2 14678.721} C_VEL
LIN {X 0,Y 301.753,Z 911.476,A -85,B 0,C 180,E1 14689.842,E2 14689.842} C_VEL
LIN {X 0,Y 309.478,Z 881.54,A -85,B 0,C 180,E1 14701.398,E2 14701.398} C_VEL
LIN {X 0,Y 324.5,Z 838.445,A -85,B 0,C 180,E1 14711.464,E2 14711.464} C_VEL
LIN {X 0,Y 336.677,Z 803.102,A -85,B 0,C 180,E1 14716.895,E2 14716.895} C_VEL
LIN {X 0,Y 339.258,Z 776.369,A -85,B 0,C 180,E1 14720.836,E2 14720.836} C_VEL
LIN {X 0,Y 354.987,Z 715.994,A -85,B 0,C 180,E1 14725.397,E2 14725.397} C_VEL
LIN {X 0,Y 356.677,Z 701.354,A -85,B 0,C 180,E1 14726.345,E2 14726.345} C_VEL
LIN {X 0,Y 340.809,Z 659.169,A -85,B 0,C 180,E1 14733.09,E2 14733.09} C_VEL
LIN {X 0,Y 323.361,Z 630.358,A -85,B 0,C 180,E1 14741.239,E2 14741.239} C_VEL
LIN {X 0,Y 314.258,Z 617.161,A -85,B 0,C 180,E1 14749.097,E2 14749.097} C_VEL
LIN {X 0,Y 313.114,Z 615.116,A -85,B 0,C 180,E1 14759.012,E2 14759.012} C_VEL
LIN {X 0,Y 318.362,Z 622.772,A -85,B 0,C 180,E1 14765.51,E2 14765.51} C_VEL
LIN {X 0,Y 331.442,Z 643.955,A -85,B 0,C 180,E1 14773.533,E2 14773.533} C_VEL
LIN {X 0,Y 346.275,Z 680.414,A -85,B 0,C 180,E1 14781.169,E2 14781.169} C_VEL
LIN {X 0,Y 347.146,Z 693.235,A -85,B 0,C 180,E1 14782.756,E2 14782.756} C_VEL
LIN {X 0,Y 332.506,Z 745.727,A -85,B 0,C 180,E1 14787.594,E2 14787.594} C_VEL
LIN {X 0,Y 316.225,Z 788.435,A -85,B 0,C 180,E1 14794.745,E2 14794.745} C_VEL
LIN {X 0,Y 302.733,Z 819.339,A -85,B 0,C 180,E1 14804.256,E2 14804.256} C_VEL
LIN {X 0,Y 296.02,Z 834.798,A -85,B 0,C 180,E1 14813.878,E2 14813.878} C_VEL
LIN {X 0,Y 293.516,Z 839.01,A -85,B 0,C 180,E1 14824.877,E2 14824.877} C_VEL
LIN {X 0,Y 296.517,Z 829.752,A -85,B 0,C 180,E1 14836.025,E2 14836.025} C_VEL
LIN {X 0,Y 304.87,Z 806.062,A -85,B 0,C 180,E1 14846.515,E2 14846.515} C_VEL
LIN {X 0,Y 317.804,Z 769.18,A -85,B 0,C 180,E1 14855.138,E2 14855.138} C_VEL
LIN {X 0,Y 331.759,Z 721.494,A -85,B 0,C 180,E1 14861.378,E2 14861.378} C_VEL
LIN {X 0,Y 339.657,Z 677.573,A -85,B 0,C 180,E1 14864.877,E2 14864.877} C_VEL
LIN {X 0,Y 320.325,Z 634.365,A -85,B 0,C 180,E1 14871.689,E2 14871.689} C_VEL
LIN {X 0,Y 292.883,Z 593.743,A -85,B 0,C 180,E1 14881.412,E2 14881.412} C_VEL
LIN {X 0,Y 288.906,Z 586.94,A -85,B 0,C 180,E1 14883.473,E2 14883.473} C_VEL
LIN {X 0,Y 288.741,Z 586.94,A -85,B 0,C 180,E1 14895.197,E2 14895.197} C_VEL
LIN {X 0,Y 288.853,Z 586.94,A -85,B 0,C 180,E1 14906.467,E2 14906.467} C_VEL
LIN {X 0,Y 289.531,Z 586.94,A -85,B 0,C 180,E1 14920.029,E2 14920.029} C_VEL
LIN {X 0,Y 290.711,Z 586.94,A -85,B 0,C 180,E1 14932.447,E2 14932.447} C_VEL
LIN {X 0,Y 290.832,Z 586.94,A -85,B 0,C 180,E1 14944.43,E2 14944.43} C_VEL
LIN {X 0,Y 290.468,Z 588.972,A -85,B 0,C 180,E1 14952.286,E2 14952.286} C_VEL
LIN {X 0,Y 320.295,Z 632.474,A -85,B 0,C 180,E1 14963.312,E2 14963.312} C_VEL
LIN {X 0,Y 347.247,Z 682.85,A -85,B 0,C 180,E1 14971.386,E2 14971.386} C_VEL
LIN {X 0,Y 354.804,Z 707.843,A -85,B 0,C 180,E1 14974.425,E2 14974.425} C_VEL
LIN {X 0,Y 340.473,Z 770.05,A -85,B 0,C 180,E1 14978.738,E2 14978.738} C_VEL
LIN {X 0,Y 322.072,Z 825.991,A -85,B 0,C 180,E1 14985.619,E2 14985.619} C_VEL
LIN {X 0,Y 305.618,Z 871.807,A -85,B 0,C 180,E1 14995.177,E2 14995.177} C_VEL
LIN {X 0,Y 295.278,Z 904.438,A -85,B 0,C 180,E1 15006.527,E2 15006.527} C_VEL
LIN {X 0,Y 292.347,Z 923.18,A -85,B 0,C 180,E1 15018.015,E2 15018.015} C_VEL
LIN {X 0,Y 292.089,Z 929.593,A -85,B 0,C 180,E1 15028.51,E2 15028.51} C_VEL
LIN {X 0,Y 292.282,Z 926.029,A -85,B 0,C 180,E1 15038.767,E2 15038.767} C_VEL
LIN {X 0,Y 293.907,Z 910.202,A -85,B 0,C 180,E1 15050.371,E2 15050.371} C_VEL
LIN {X 0,Y 302.285,Z 880.149,A -85,B 0,C 180,E1 15062.233,E2 15062.233} C_VEL
LIN {X 0,Y 318.41,Z 836.224,A -85,B 0,C 180,E1 15072.613,E2 15072.613} C_VEL
LIN {X 0,Y 337.265,Z 782.842,A -85,B 0,C 180,E1 15080.148,E2 15080.148} C_VEL
LIN {X 0,Y 339.258,Z 776.369,A -85,B 0,C 180,E1 15080.836,E2 15080.836} C_VEL
LIN {X 0,Y 341.86,Z 747.802,A -85,B 0,C 180,E1 15084.368,E2 15084.368} C_VEL
LIN {X 0,Y 351.169,Z 704.537,A -85,B 0,C 180,E1 15087.192,E2 15087.192} C_VEL
LIN {X 0,Y 336.764,Z 664.039,A -85,B 0,C 180,E1 15093.99,E2 15093.99} C_VEL
LIN {X 0,Y 320.703,Z 636.596,A -85,B 0,C 180,E1 15102.238,E2 15102.238} C_VEL
LIN {X 0,Y 312.886,Z 624.839,A -85,B 0,C 180,E1 15109.579,E2 15109.579} C_VEL
LIN {X 0,Y 312.104,Z 623.247,A -85,B 0,C 180,E1 15119.183,E2 15119.183} C_VEL
LIN {X 0,Y 318.525,Z 632.514,A -85,B 0,C 180,E1 15126.56,E2 15126.56} C_VEL
LIN {X 0,Y 332.521,Z 659.455,A -85,B 0,C 180,E1 15135.259,E2 15135.259} C_VEL
LIN {X 0,Y 342.437,Z 693.084,A -85,B 0,C 180,E1 15141.653,E2 15141.653} C_VEL
LIN {X 0,Y 326.94,Z 746.603,A -85,B 0,C 180,E1 15146.588,E2 15146.588} C_VEL
LIN {X 0,Y 309.496,Z 790.233,A -85,B 0,C 180,E1 15154.024,E2 15154.024} C_VEL
LIN {X 0,Y 295.878,Z 819.679,A -85,B 0,C 180,E1 15163.205,E2 15163.205} C_VEL
LIN {X 0,Y 288.588,Z 835.333,A -85,B 0,C 180,E1 15172.793,E2 15172.793} C_VEL
LIN {X 0,Y 285.628,Z 840.468,A -85,B 0,C 180,E1 15183.155,E2 15183.155} C_VEL
LIN {X 0,Y 287.983,Z 833.128,A -85,B 0,C 180,E1 15194.725,E2 15194.725} C_VEL
LIN {X 0,Y 295.721,Z 811.762,A -85,B 0,C 180,E1 15205.587,E2 15205.587} C_VEL
LIN {X 0,Y 308.507,Z 777.512,A -85,B 0,C 180,E1 15214.586,E2 15214.586} C_VEL
LIN {X 0,Y 323.635,Z 730.14,A -85,B 0,C 180,E1 15221.496,E2 15221.496} C_VEL
LIN {X 0,Y 333.916,Z 681.302,A -85,B 0,C 180,E1 15225.598,E2 15225.598} C_VEL
LIN {X 0,Y 315.381,Z 638.614,A -85,B 0,C 180,E1 15232.651,E2 15232.651} C_VEL
LIN {X 0,Y 289.47,Z 600.336,A -85,B 0,C 180,E1 15242.25,E2 15242.25} C_VEL
LIN {X 0,Y 280.783,Z 586.94,A -85,B 0,C 180,E1 15246.623,E2 15246.623} C_VEL
LIN {X 0,Y 280.614,Z 586.94,A -85,B 0,C 180,E1 15257.41,E2 15257.41} C_VEL
LIN {X 0,Y 280.855,Z 586.94,A -85,B 0,C 180,E1 15269.061,E2 15269.061} C_VEL
LIN {X 0,Y 281.769,Z 586.94,A -85,B 0,C 180,E1 15282.715,E2 15282.715} C_VEL
LIN {X 0,Y 282.791,Z 586.94,A -85,B 0,C 180,E1 15295.326,E2 15295.326} C_VEL
LIN {X 0,Y 282.636,Z 586.94,A -85,B 0,C 180,E1 15306.627,E2 15306.627} C_VEL
LIN {X 0,Y 282.71,Z 589.082,A -85,B 0,C 180,E1 15309.108,E2 15309.108} C_VEL
LIN {X 0,Y 309.348,Z 627.005,A -85,B 0,C 180,E1 15320.205,E2 15320.205} C_VEL
LIN {X 0,Y 337.662,Z 677.28,A -85,B 0,C 180,E1 15329.232,E2 15329.232} C_VEL
LIN {X 0,Y 348.751,Z 710.164,A -85,B 0,C 180,E1 15333.602,E2 15333.602} C_VEL
LIN {X 0,Y 333.501,Z 772.769,A -85,B 0,C 180,E1 15338.117,E2 15338.117} C_VEL
LIN {X 0,Y 314.856,Z 826.945,A -85,B 0,C 180,E1 15345.023,E2 15345.023} C_VEL
LIN {X 0,Y 297.627,Z 872.832,A -85,B 0,C 180,E1 15354.996,E2 15354.996} C_VEL
LIN {X 0,Y 287.179,Z 904.735,A -85,B 0,C 180,E1 15366.65,E2 15366.65} C_VEL
LIN {X 0,Y 284.404,Z 921.898,A -85,B 0,C 180,E1 15377.675,E2 15377.675} C_VEL
LIN {X 0,Y 284.174,Z 928.374,A -85,B 0,C 180,E1 15388.469,E2 15388.469} C_VEL
LIN {X 0,Y 284.327,Z 924.233,A -85,B 0,C 180,E1 15399.607,E2 15399.607} C_VEL
LIN {X 0,Y 286.545,Z 907.179,A -85,B 0,C 180,E1 15411.832,E2 15411.832} C_VEL
LIN {X 0,Y 296.618,Z 875.058,A -85,B 0,C 180,E1 15424.246,E2 15424.246} C_VEL
LIN {X 0,Y 314.4,Z 828.913,A -85,B 0,C 180,E1 15434.739,E2 15434.739} C_VEL
LIN {X 0,Y 334.632,Z 772.691,A -85,B 0,C 180,E1 15442.162,E2 15442.162} C_VEL
LIN {X 0,Y 341.86,Z 747.802,A -85,B 0,C 180,E1 15444.368,E2 15444.368} C_VEL
LIN {X 0,Y 344.512,Z 717.37,A -85,B 0,C 180,E1 15447.361,E2 15447.361} C_VEL
LIN {X 0,Y 345.1,Z 704.809,A -85,B 0,C 180,E1 15448.476,E2 15448.476} C_VEL
LIN {X 0,Y 331.437,Z 666.274,A -85,B 0,C 180,E1 15455.55,E2 15455.55} C_VEL
LIN {X 0,Y 316.681,Z 639.865,A -85,B 0,C 180,E1 15464.423,E2 15464.423} C_VEL
LIN {X 0,Y 310.94,Z 631.66,A -85,B 0,C 180,E1 15471.285,E2 15471.285} C_VEL
LIN {X 0,Y 311.367,Z 631.765,A -85,B 0,C 180,E1 15479.914,E2 15479.914} C_VEL
LIN {X 0,Y 317.656,Z 642.409,A -85,B 0,C 180,E1 15487.045,E2 15487.045} C_VEL
LIN {X 0,Y 329.58,Z 667.419,A -85,B 0,C 180,E1 15495.057,E2 15495.057} C_VEL
LIN {X 0,Y 337.029,Z 696.857,A -85,B 0,C 180,E1 15500.777,E2 15500.777} C_VEL
LIN {X 0,Y 320.746,Z 749.544,A -85,B 0,C 180,E1 15505.82,E2 15505.82} C_VEL
LIN {X 0,Y 302.528,Z 792.713,A -85,B 0,C 180,E1 15513.435,E2 15513.435} C_VEL
LIN {X 0,Y 287.648,Z 823.057,A -85,B 0,C 180,E1 15523.543,E2 15523.543} C_VEL
LIN {X 0,Y 279.679,Z 839.061,A -85,B 0,C 180,E1 15535.271,E2 15535.271} C_VEL
LIN {X 0,Y 277.773,Z 841.271,A -85,B 0,C 180,E1 15545.813,E2 15545.813} C_VEL
LIN {X 0,Y 281.641,Z 830.463,A -85,B 0,C 180,E1 15557.775,E2 15557.775} C_VEL
LIN {X 0,Y 291.309,Z 806.017,A -85,B 0,C 180,E1 15568.509,E2 15568.509} C_VEL
LIN {X 0,Y 305.371,Z 769.065,A -85,B 0,C 180,E1 15577.138,E2 15577.138} C_VEL
LIN {X 0,Y 320.503,Z 720.758,A -85,B 0,C 180,E1 15583.46,E2 15583.46} C_VEL
LIN {X 0,Y 327.62,Z 683.077,A -85,B 0,C 180,E1 15586.623,E2 15586.623} C_VEL
LIN {X 0,Y 309.595,Z 641.353,A -85,B 0,C 180,E1 15593.949,E2 15593.949} C_VEL
LIN {X 0,Y 285.484,Z 605.807,A -85,B 0,C 180,E1 15603.42,E2 15603.42} C_VEL
LIN {X 0,Y 272.527,Z 586.94,A -85,B 0,C 180,E1 15611.194,E2 15611.194} C_VEL
LIN {X 0,Y 272.619,Z 586.94,A -85,B 0,C 180,E1 15624.175,E2 15624.175} C_VEL
LIN {X 0,Y 273.176,Z 586.94,A -85,B 0,C 180,E1 15636.436,E2 15636.436} C_VEL
LIN {X 0,Y 274.344,Z 586.94,A -85,B 0,C 180,E1 15648.78,E2 15648.78} C_VEL
LIN {X 0,Y 275.293,Z 586.94,A -85,B 0,C 180,E1 15661.518,E2 15661.518} C_VEL
LIN {X 0,Y 274.962,Z 589.012,A -85,B 0,C 180,E1 15665.416,E2 15665.416} C_VEL
LIN {X 0,Y 298.604,Z 622.143,A -85,B 0,C 180,E1 15676.764,E2 15676.764} C_VEL
LIN {X 0,Y 326.364,Z 668.585,A -85,B 0,C 180,E1 15686.332,E2 15686.332} C_VEL
LIN {X 0,Y 342.862,Z 711.967,A -85,B 0,C 180,E1 15692.738,E2 15692.738} C_VEL
LIN {X 0,Y 326.588,Z 775.451,A -85,B 0,C 180,E1 15697.468,E2 15697.468} C_VEL
LIN {X 0,Y 306.649,Z 830.758,A -85,B 0,C 180,E1 15704.896,E2 15704.896} C_VEL
LIN {X 0,Y 288.947,Z 875.852,A -85,B 0,C 180,E1 15715.402,E2 15715.402} C_VEL
LIN {X 0,Y 278.937,Z 905.641,A -85,B 0,C 180,E1 15727.156,E2 15727.156} C_VEL
LIN {X 0,Y 276.445,Z 922.208,A -85,B 0,C 180,E1 15738.921,E2 15738.921} C_VEL
LIN {X 0,Y 276.281,Z 927.151,A -85,B 0,C 180,E1 15748.425,E2 15748.425} C_VEL
LIN {X 0,Y 276.407,Z 922.992,A -85,B 0,C 180,E1 15759.885,E2 15759.885} C_VEL
LIN {X 0,Y 278.508,Z 907.12,A -85,B 0,C 180,E1 15771.809,E2 15771.809} C_VEL
LIN {X 0,Y 288.878,Z 875.606,A -85,B 0,C 180,E1 15784.611,E2 15784.611} C_VEL
LIN {X 0,Y 307.85,Z 828.808,A -85,B 0,C 180,E1 15795.622,E2 15795.622} C_VEL
LIN {X 0,Y 328.861,Z 773.026,A -85,B 0,C 180,E1 15803.126,E2 15803.126} C_VEL
LIN {X 0,Y 344.512,Z 717.37,A -85,B 0,C 180,E1 15807.361,E2 15807.361} C_VEL
LIN {X 0,Y 342.677,Z 709.13,A -85,B 0,C 180,E1 15808.624,E2 15808.624} C_VEL
LIN {X 0,Y 338.353,Z 702.246,A -85,B 0,C 180,E1 15810.313,E2 15810.313} C_VEL
LIN {X 0,Y 325.616,Z 667.31,A -85,B 0,C 180,E1 15817.562,E2 15817.562} C_VEL
LIN {X 0,Y 313.828,Z 646.129,A -85,B 0,C 180,E1 15825.801,E2 15825.801} C_VEL
LIN {X 0,Y 309.304,Z 638.628,A -85,B 0,C 180,E1 15833.011,E2 15833.011} C_VEL
LIN {X 0,Y 311.545,Z 641.157,A -85,B 0,C 180,E1 15842.006,E2 15842.006} C_VEL
LIN {X 0,Y 321.822,Z 662.913,A -85,B 0,C 180,E1 15851.576,E2 15851.576} C_VEL
LIN {X 0,Y 332.229,Z 697.771,A -85,B 0,C 180,E1 15859.625,E2 15859.625} C_VEL
LIN {X 0,Y 315.313,Z 750.697,A -85,B 0,C 180,E1 15864.767,E2 15864.767} C_VEL
LIN {X 0,Y 296.466,Z 793.394,A -85,B 0,C 180,E1 15872.375,E2 15872.375} C_VEL
LIN {X 0,Y 280.686,Z 823.756,A -85,B 0,C 180,E1 15882.576,E2 15882.576} C_VEL
LIN {X 0,Y 272.194,Z 839.76,A -85,B 0,C 180,E1 15894.171,E2 15894.171} C_VEL
LIN {X 0,Y 269.806,Z 842.665,A -85,B 0,C 180,E1 15905.051,E2 15905.051} C_VEL
LIN {X 0,Y 273.106,Z 833.773,A -85,B 0,C 180,E1 15916.671,E2 15916.671} C_VEL
LIN {X 0,Y 282.702,Z 810.402,A -85,B 0,C 180,E1 15928.09,E2 15928.09} C_VEL
LIN {X 0,Y 297.49,Z 773.88,A -85,B 0,C 180,E1 15937.328,E2 15937.328} C_VEL
LIN {X 0,Y 313.255,Z 726.451,A -85,B 0,C 180,E1 15943.948,E2 15943.948} C_VEL
LIN {X 0,Y 321.684,Z 685.984,A -85,B 0,C 180,E1 15947.508,E2 15947.508} C_VEL
LIN {X 0,Y 303.741,Z 643.772,A -85,B 0,C 180,E1 15955.343,E2 15955.343} C_VEL
LIN {X 0,Y 279.822,Z 608.31,A -85,B 0,C 180,E1 15965.544,E2 15965.544} C_VEL
LIN {X 0,Y 266.176,Z 591.839,A -85,B 0,C 180,E1 15973.818,E2 15973.818} C_VEL
LIN {X 0,Y 264.507,Z 586.94,A -85,B 0,C 180,E1 15975.821,E2 15975.821} C_VEL
LIN {X 0,Y 264.632,Z 586.94,A -85,B 0,C 180,E1 15986.931,E2 15986.931} C_VEL
LIN {X 0,Y 265.396,Z 586.94,A -85,B 0,C 180,E1 16000.645,E2 16000.645} C_VEL
LIN {X 0,Y 266.595,Z 586.94,A -85,B 0,C 180,E1 16011.759,E2 16011.759} C_VEL
LIN {X 0,Y 267.491,Z 588.995,A -85,B 0,C 180,E1 16021.157,E2 16021.157} C_VEL
LIN {X 0,Y 287.895,Z 617.368,A -85,B 0,C 180,E1 16032.794,E2 16032.794} C_VEL
LIN {X 0,Y 315.143,Z 660.749,A -85,B 0,C 180,E1 16043.246,E2 16043.246} C_VEL
LIN {X 0,Y 335.872,Z 708.985,A -85,B 0,C 180,E1 16051.233,E2 16051.233} C_VEL
LIN {X 0,Y 334.939,Z 722.581,A -85,B 0,C 180,E1 16052.336,E2 16052.336} C_VEL
LIN {X 0,Y 317.312,Z 784.637,A -85,B 0,C 180,E1 16057.507,E2 16057.507} C_VEL
LIN {X 0,Y 296.957,Z 837.749,A -85,B 0,C 180,E1 16065.436,E2 16065.436} C_VEL
LIN {X 0,Y 279.985,Z 879.022,A -85,B 0,C 180,E1 16075.967,E2 16075.967} C_VEL
LIN {X 0,Y 270.389,Z 908.06,A -85,B 0,C 180,E1 16088.603,E2 16088.603} C_VEL
LIN {X 0,Y 268.38,Z 923.009,A -85,B 0,C 180,E1 16101.13,E2 16101.13} C_VEL
LIN {X 0,Y 268.509,Z 925.907,A -85,B 0,C 180,E1 16111.618,E2 16111.618} C_VEL
LIN {X 0,Y 268.569,Z 919.062,A -85,B 0,C 180,E1 16123.061,E2 16123.061} C_VEL
LIN {X 0,Y 273.854,Z 896.434,A -85,B 0,C 180,E1 16137.202,E2 16137.202} C_VEL
LIN {X 0,Y 288.591,Z 858.833,A -85,B 0,C 180,E1 16149.965,E2 16149.965} C_VEL
LIN {X 0,Y 309.043,Z 810.265,A -85,B 0,C 180,E1 16159.56,E2 16159.56} C_VEL
LIN {X 0,Y 329.791,Z 752.84,A -85,B 0,C 180,E1 16166.023,E2 16166.023} C_VEL
LIN {X 0,Y 340.321,Z 710.348,A -85,B 0,C 180,E1 16169.035,E2 16169.035} C_VEL
LIN {X 0,Y 338.353,Z 702.246,A -85,B 0,C 180,E1 16170.313,E2 16170.313} C_VEL
LIN {X 0,Y 326.989,Z 684.955,A -85,B 0,C 180,E1 16175.334,E2 16175.334} C_VEL
LIN {X 0,Y 314.903,Z 658.735,A -85,B 0,C 180,E1 16183.525,E2 16183.525} C_VEL
LIN {X 0,Y 308.774,Z 647.774,A -85,B 0,C 180,E1 16191.045,E2 16191.045} C_VEL
LIN {X 0,Y 308.751,Z 647.393,A -85,B 0,C 180,E1 16199.526,E2 16199.526} C_VEL
LIN {X 0,Y 315.133,Z 660.857,A -85,B 0,C 180,E1 16207.934,E2 16207.934} C_VEL
LIN {X 0,Y 324.493,Z 688.654,A -85,B 0,C 180,E1 16215.995,E2 16215.995} C_VEL
LIN {X 0,Y 326.089,Z 705.226,A -85,B 0,C 180,E1 16219.004,E2 16219.004} C_VEL
LIN {X 0,Y 308.097,Z 756.655,A -85,B 0,C 180,E1 16224.33,E2 16224.33} C_VEL
LIN {X 0,Y 288.47,Z 798.023,A -85,B 0,C 180,E1 16232.295,E2 16232.295} C_VEL
LIN {X 0,Y 272.218,Z 827.555,A -85,B 0,C 180,E1 16243.143,E2 16243.143} C_VEL
LIN {X 0,Y 263.959,Z 841.783,A -85,B 0,C 180,E1 16254.911,E2 16254.911} C_VEL
LIN {X 0,Y 262.187,Z 842.929,A -85,B 0,C 180,E1 16267.902,E2 16267.902} C_VEL
LIN {X 0,Y 267.283,Z 830.346,A -85,B 0,C 180,E1 16280.195,E2 16280.195} C_VEL
LIN {X 0,Y 279.12,Z 803.021,A -85,B 0,C 180,E1 16291.559,E2 16291.559} C_VEL
LIN {X 0,Y 295.695,Z 762.653,A -85,B 0,C 180,E1 16300.349,E2 16300.349} C_VEL
LIN {X 0,Y 311.889,Z 711.649,A -85,B 0,C 180,E1 16306.429,E2 16306.429} C_VEL
LIN {X 0,Y 315.899,Z 689.208,A -85,B 0,C 180,E1 16308.377,E2 16308.377} C_VEL
LIN {X 0,Y 298.818,Z 648.14,A -85,B 0,C 180,E1 16316.429,E2 16316.429} C_VEL
LIN {X 0,Y 276.913,Z 615.045,A -85,B 0,C 180,E1 16326.357,E2 16326.357} C_VEL
LIN {X 0,Y 260.889,Z 594.075,A -85,B 0,C 180,E1 16337.264,E2 16337.264} C_VEL
LIN {X 0,Y 256.476,Z 586.94,A -85,B 0,C 180,E1 16343.015,E2 16343.015} C_VEL
LIN {X 0,Y 257.072,Z 586.94,A -85,B 0,C 180,E1 16357.377,E2 16357.377} C_VEL
LIN {X 0,Y 258.532,Z 586.94,A -85,B 0,C 180,E1 16371.5,E2 16371.5} C_VEL
LIN {X 0,Y 259.199,Z 589.527,A -85,B 0,C 180,E1 16375.106,E2 16375.106} C_VEL
LIN {X 0,Y 266.818,Z 599.007,A -85,B 0,C 180,E1 16381.567,E2 16381.567} C_VEL
LIN {X 0,Y 285.673,Z 624.901,A -85,B 0,C 180,E1 16392.333,E2 16392.333} C_VEL
LIN {X 0,Y 311.159,Z 666.664,A -85,B 0,C 180,E1 16402.579,E2 16402.579} C_VEL
LIN {X 0,Y 330.57,Z 714.185,A -85,B 0,C 180,E1 16410.712,E2 16410.712} C_VEL
LIN {X 0,Y 314.15,Z 776.441,A -85,B 0,C 180,E1 16415.687,E2 16415.687} C_VEL
LIN {X 0,Y 293.411,Z 829.661,A -85,B 0,C 180,E1 16423.066,E2 16423.066} C_VEL
LIN {X 0,Y 274.175,Z 874.475,A -85,B 0,C 180,E1 16433.979,E2 16433.979} C_VEL
LIN {X 0,Y 263.1,Z 904.472,A -85,B 0,C 180,E1 16446.682,E2 16446.682} C_VEL
LIN {X 0,Y 260.566,Z 919.653,A -85,B 0,C 180,E1 16458.237,E2 16458.237} C_VEL
LIN {X 0,Y 260.445,Z 924.701,A -85,B 0,C 180,E1 16468.329,E2 16468.329} C_VEL
LIN {X 0,Y 260.541,Z 920.884,A -85,B 0,C 180,E1 16480.062,E2 16480.062} C_VEL
LIN {X 0,Y 263.157,Z 904.234,A -85,B 0,C 180,E1 16493.323,E2 16493.323} C_VEL
LIN {X 0,Y 275.385,Z 872.201,A -85,B 0,C 180,E1 16506.849,E2 16506.849} C_VEL
LIN {X 0,Y 296.172,Z 825.947,A -85,B 0,C 180,E1 16517.981,E2 16517.981} C_VEL
LIN {X 0,Y 318.98,Z 770.07,A -85,B 0,C 180,E1 16525.522,E2 16525.522} C_VEL
LIN {X 0,Y 334.833,Z 712.913,A -85,B 0,C 180,E1 16530.057,E2 16530.057} C_VEL
LIN {X 0,Y 326.989,Z 684.955,A -85,B 0,C 180,E1 16535.334,E2 16535.334} C_VEL
LIN {X 0,Y 318.652,Z 678.956,A -85,B 0,C 180,E1 16539.185,E2 16539.185} C_VEL
LIN {X 0,Y 309.167,Z 659.049,A -85,B 0,C 180,E1 16547.849,E2 16547.849} C_VEL
LIN {X 0,Y 306.711,Z 653.958,A -85,B 0,C 180,E1 16557.751,E2 16557.751} C_VEL
LIN {X 0,Y 310.68,Z 663.65,A -85,B 0,C 180,E1 16565.48,E2 16565.48} C_VEL
LIN {X 0,Y 318.593,Z 687.34,A -85,B 0,C 180,E1 16573.65,E2 16573.65} C_VEL
LIN {X 0,Y 321.375,Z 707.448,A -85,B 0,C 180,E1 16577.921,E2 16577.921} C_VEL
LIN {X 0,Y 302.362,Z 758.971,A -85,B 0,C 180,E1 16583.374,E2 16583.374} C_VEL
LIN {X 0,Y 281.548,Z 800.612,A -85,B 0,C 180,E1 16591.651,E2 16591.651} C_VEL
LIN {X 0,Y 265.426,Z 828.119,A -85,B 0,C 180,E1 16602,E2 16602} C_VEL
LIN {X 0,Y 256.911,Z 841.958,A -85,B 0,C 180,E1 16612.961,E2 16612.961} C_VEL
LIN {X 0,Y 254.006,Z 845.42,A -85,B 0,C 180,E1 16623.381,E2 16623.381} C_VEL
LIN {X 0,Y 256.875,Z 838.065,A -85,B 0,C 180,E1 16635.828,E2 16635.828} C_VEL
LIN {X 0,Y 265.975,Z 817.539,A -85,B 0,C 180,E1 16647.637,E2 16647.637} C_VEL
LIN {X 0,Y 281.561,Z 782.948,A -85,B 0,C 180,E1 16657.745,E2 16657.745} C_VEL
LIN {X 0,Y 299.442,Z 735.392,A -85,B 0,C 180,E1 16665.21,E2 16665.21} C_VEL
LIN {X 0,Y 310.099,Z 692.454,A -85,B 0,C 180,E1 16669.289,E2 16669.289} C_VEL
LIN {X 0,Y 293.928,Z 652.183,A -85,B 0,C 180,E1 16677.586,E2 16677.586} C_VEL
LIN {X 0,Y 273.18,Z 620.575,A -85,B 0,C 180,E1 16687.663,E2 16687.663} C_VEL
LIN {X 0,Y 258.429,Z 601.245,A -85,B 0,C 180,E1 16698.385,E2 16698.385} C_VEL
LIN {X 0,Y 252.51,Z 593.867,A -85,B 0,C 180,E1 16705.7,E2 16705.7} C_VEL
LIN {X 0,Y 249.881,Z 589.419,A -85,B 0,C 180,E1 16721.837,E2 16721.837} C_VEL
LIN {X 0,Y 257.778,Z 597.449,A -85,B 0,C 180,E1 16734.766,E2 16734.766} C_VEL
LIN {X 0,Y 268.187,Z 609.979,A -85,B 0,C 180,E1 16743.275,E2 16743.275} C_VEL
LIN {X 0,Y 291.45,Z 644.638,A -85,B 0,C 180,E1 16755.446,E2 16755.446} C_VEL
LIN {X 0,Y 314.22,Z 688.22,A -85,B 0,C 180,E1 16764.929,E2 16764.929} C_VEL
LIN {X 0,Y 324.354,Z 720.903,A -85,B 0,C 180,E1 16770.195,E2 16770.195} C_VEL
LIN {X 0,Y 306.446,Z 781.152,A -85,B 0,C 180,E1 16775.204,E2 16775.204} C_VEL
LIN {X 0,Y 285.032,Z 833.387,A -85,B 0,C 180,E1 16782.939,E2 16782.939} C_VEL
LIN {X 0,Y 265.695,Z 876.516,A -85,B 0,C 180,E1 16794.166,E2 16794.166} C_VEL
LIN {X 0,Y 254.881,Z 905.225,A -85,B 0,C 180,E1 16807.23,E2 16807.23} C_VEL
LIN {X 0,Y 252.605,Z 919.748,A -85,B 0,C 180,E1 16819.616,E2 16819.616} C_VEL
LIN {X 0,Y 252.664,Z 923.46,A -85,B 0,C 180,E1 16831.719,E2 16831.719} C_VEL
LIN {X 0,Y 252.789,Z 916.569,A -85,B 0,C 180,E1 16843.892,E2 16843.892} C_VEL
LIN {X 0,Y 258.91,Z 893.816,A -85,B 0,C 180,E1 16858.915,E2 16858.915} C_VEL
LIN {X 0,Y 275.926,Z 855.515,A -85,B 0,C 180,E1 16872.427,E2 16872.427} C_VEL
LIN {X 0,Y 299.04,Z 805.843,A -85,B 0,C 180,E1 16882.288,E2 16882.288} C_VEL
LIN {X 0,Y 321.785,Z 746.346,A -85,B 0,C 180,E1 16888.797,E2 16888.797} C_VEL
LIN {X 0,Y 329.654,Z 716.366,A -85,B 0,C 180,E1 16890.977,E2 16890.977} C_VEL
LIN {X 0,Y 319.846,Z 681.867,A -85,B 0,C 180,E1 16898.317,E2 16898.317} C_VEL
LIN {X 0,Y 318.652,Z 678.956,A -85,B 0,C 180,E1 16899.185,E2 16899.185} C_VEL
LIN {X 0,Y 311.393,Z 675.586,A -85,B 0,C 180,E1 16903.301,E2 16903.301} C_VEL
LIN {X 0,Y 305.536,Z 663.213,A -85,B 0,C 180,E1 16911.507,E2 16911.507} C_VEL
LIN {X 0,Y 305.482,Z 663.272,A -85,B 0,C 180,E1 16919.699,E2 16919.699} C_VEL
LIN {X 0,Y 310.784,Z 678.413,A -85,B 0,C 180,E1 16928.386,E2 16928.386} C_VEL
LIN {X 0,Y 317.052,Z 708.584,A -85,B 0,C 180,E1 16936.696,E2 16936.696} C_VEL
LIN {X 0,Y 296.809,Z 761.144,A -85,B 0,C 180,E1 16942.354,E2 16942.354} C_VEL
LIN {X 0,Y 275.447,Z 801.746,A -85,B 0,C 180,E1 16950.563,E2 16950.563} C_VEL
LIN {X 0,Y 257.733,Z 830.302,A -85,B 0,C 180,E1 16961.723,E2 16961.723} C_VEL
LIN {X 0,Y 248.315,Z 844.511,A -85,B 0,C 180,E1 16974.511,E2 16974.511} C_VEL
LIN {X 0,Y 246.163,Z 846.038,A -85,B 0,C 180,E1 16986.379,E2 16986.379} C_VEL
LIN {X 0,Y 250.968,Z 835.039,A -85,B 0,C 180,E1 16999.55,E2 16999.55} C_VEL
LIN {X 0,Y 263.111,Z 809.877,A -85,B 0,C 180,E1 17011.654,E2 17011.654} C_VEL
LIN {X 0,Y 280.459,Z 771.636,A -85,B 0,C 180,E1 17021.115,E2 17021.115} C_VEL
LIN {X 0,Y 298.308,Z 722.087,A -85,B 0,C 180,E1 17027.773,E2 17027.773} C_VEL
LIN {X 0,Y 304.162,Z 695.159,A -85,B 0,C 180,E1 17030.328,E2 17030.328} C_VEL
LIN {X 0,Y 288.985,Z 656.285,A -85,B 0,C 180,E1 17038.781,E2 17038.781} C_VEL
LIN {X 0,Y 268.158,Z 623.437,A -85,B 0,C 180,E1 17049.955,E2 17049.955} C_VEL
LIN {X 0,Y 255.512,Z 607.606,A -85,B 0,C 180,E1 17060.169,E2 17060.169} C_VEL
LIN {X 0,Y 251.17,Z 601.647,A -85,B 0,C 180,E1 17066.071,E2 17066.071} C_VEL
LIN {X 0,Y 248.772,Z 597.315,A -85,B 0,C 180,E1 17081.652,E2 17081.652} C_VEL
LIN {X 0,Y 256.37,Z 605.314,A -85,B 0,C 180,E1 17094.418,E2 17094.418} C_VEL
LIN {X 0,Y 266.596,Z 618.221,A -85,B 0,C 180,E1 17102.992,E2 17102.992} C_VEL
LIN {X 0,Y 288.754,Z 651.723,A -85,B 0,C 180,E1 17114.919,E2 17114.919} C_VEL
LIN {X 0,Y 310.074,Z 694.882,A -85,B 0,C 180,E1 17124.513,E2 17124.513} C_VEL
LIN {X 0,Y 318.292,Z 724.067,A -85,B 0,C 180,E1 17129.319,E2 17129.319} C_VEL
LIN {X 0,Y 298.759,Z 785.695,A -85,B 0,C 180,E1 17134.691,E2 17134.691} C_VEL
LIN {X 0,Y 276.172,Z 838.111,A -85,B 0,C 180,E1 17143.03,E2 17143.03} C_VEL
LIN {X 0,Y 256.153,Z 880.819,A -85,B 0,C 180,E1 17155.233,E2 17155.233} C_VEL
LIN {X 0,Y 246.265,Z 907.91,A -85,B 0,C 180,E1 17169.267,E2 17169.267} C_VEL
LIN {X 0,Y 244.606,Z 919.679,A -85,B 0,C 180,E1 17181.076,E2 17181.076} C_VEL
LIN {X 0,Y 244.738,Z 922.238,A -85,B 0,C 180,E1 17191.775,E2 17191.775} C_VEL
LIN {X 0,Y 244.918,Z 915.332,A -85,B 0,C 180,E1 17204.348,E2 17204.348} C_VEL
LIN {X 0,Y 251.824,Z 891.762,A -85,B 0,C 180,E1 17220.232,E2 17220.232} C_VEL
LIN {X 0,Y 270.367,Z 852.662,A -85,B 0,C 180,E1 17234.078,E2 17234.078} C_VEL
LIN {X 0,Y 295.16,Z 801.945,A -85,B 0,C 180,E1 17243.949,E2 17243.949} C_VEL
LIN {X 0,Y 318.04,Z 743.362,A -85,B 0,C 180,E1 17250.196,E2 17250.196} C_VEL
LIN {X 0,Y 324.495,Z 719.594,A -85,B 0,C 180,E1 17251.973,E2 17251.973} C_VEL
LIN {X 0,Y 315.714,Z 686.396,A -85,B 0,C 180,E1 17259.482,E2 17259.482} C_VEL
LIN {X 0,Y 311.393,Z 675.586,A -85,B 0,C 180,E1 17263.301,E2 17263.301} C_VEL
LIN {X 0,Y 305.968,Z 672.172,A -85,B 0,C 180,E1 17268.082,E2 17268.082} C_VEL
LIN {X 0,Y 304.486,Z 672.096,A -85,B 0,C 180,E1 17269.77,E2 17269.77} C_VEL
LIN {X 0,Y 303.26,Z 670.464,A -85,B 0,C 180,E1 17278.801,E2 17278.801} C_VEL
LIN {X 0,Y 307.08,Z 683.548,A -85,B 0,C 180,E1 17287.148,E2 17287.148} C_VEL
LIN {X 0,Y 311.995,Z 710.371,A -85,B 0,C 180,E1 17295.204,E2 17295.204} C_VEL
LIN {X 0,Y 291.446,Z 763.201,A -85,B 0,C 180,E1 17301.271,E2 17301.271} C_VEL
LIN {X 0,Y 268.559,Z 804.574,A -85,B 0,C 180,E1 17309.906,E2 17309.906} C_VEL
LIN {X 0,Y 249.896,Z 832.697,A -85,B 0,C 180,E1 17321.581,E2 17321.581} C_VEL
LIN {X 0,Y 240.946,Z 845.333,A -85,B 0,C 180,E1 17333.252,E2 17333.252} C_VEL
LIN {X 0,Y 238.38,Z 846.841,A -85,B 0,C 180,E1 17347.505,E2 17347.505} C_VEL
LIN {X 0,Y 244.021,Z 834.805,A -85,B 0,C 180,E1 17361.058,E2 17361.058} C_VEL
LIN {X 0,Y 257.52,Z 807.983,A -85,B 0,C 180,E1 17373.493,E2 17373.493} C_VEL
LIN {X 0,Y 276.087,Z 768.508,A -85,B 0,C 180,E1 17382.904,E2 17382.904} C_VEL
LIN {X 0,Y 294.44,Z 717.784,A -85,B 0,C 180,E1 17389.378,E2 17389.378} C_VEL
LIN {X 0,Y 298.465,Z 698.533,A -85,B 0,C 180,E1 17391.264,E2 17391.264} C_VEL
LIN {X 0,Y 284.148,Z 660.405,A -85,B 0,C 180,E1 17399.994,E2 17399.994} C_VEL
LIN {X 0,Y 265.347,Z 630.122,A -85,B 0,C 180,E1 17410.931,E2 17410.931} C_VEL
LIN {X 0,Y 253.6,Z 614.749,A -85,B 0,C 180,E1 17421.009,E2 17421.009} C_VEL
LIN {X 0,Y 249.347,Z 609.118,A -85,B 0,C 180,E1 17427.361,E2 17427.361} C_VEL
LIN {X 0,Y 247.719,Z 605.344,A -85,B 0,C 180,E1 17441.723,E2 17441.723} C_VEL
LIN {X 0,Y 255.049,Z 613.281,A -85,B 0,C 180,E1 17454.174,E2 17454.174} C_VEL
LIN {X 0,Y 265.037,Z 626.261,A -85,B 0,C 180,E1 17462.704,E2 17462.704} C_VEL
